	2: (* === Check loop *)
		IF NOT (MB_Lock OR MB_Start) THEN
			WHILE VarCnt<=(VARS_Max-1) AND VarSta=2 DO
				(* Check only active vars *)
				IF VARS[VarCnt].Variable<>0 THEN
					(* Check var auto-refresh on timer checks *)
					IF VARS[VarCnt].Refresh_Time>0 AND VARS[VarCnt].Refresh_Cnt=0 THEN
						VARS[VarCnt].Refresh_Cnt:=VARS[VarCnt].Refresh_Time;
						VarSta:=3;
					END_IF
					(* Check refresh for change or request *)
					CASE VARS[VarCnt].FunCode OF
						5,6,15,16: (* Write functions *)
							IF VARS[VarCnt].Variable_Size=1 THEN
								IF VARS[VarCnt].Variable^[0]<>VARS[VarCnt].Variable_Mirror THEN
									VARS[VarCnt].Variable_Mirror:=VARS[VarCnt].Variable^[0];
									VarSta:=3;
								END_IF
							ELSE
								IF VARS[VarCnt].Variable_Mirror<>0 THEN
									VARS[VarCnt].Variable_Mirror:=0;
									VarSta:=3;
								END_IF
							END_IF
						1,2,3,4: (* Write functions *)
							IF VARS[VarCnt].Variable_Mirror<>0 THEN
								VARS[VarCnt].Variable_Mirror:=0;
								VarSta:=3;
							END_IF
					END_CASE
				END_IF
				(* Process query *)
				IF VarSta=3 THEN
					MB_Lock:=TRUE;
					MB_MASTER.bUNIT_ID:=VARS[VarCnt].SlaveAddress;
					MB_MASTER.bFUNCTION_CODE:=VARS[VarCnt].FunCode;
					CASE VARS[VarCnt].FunCode OF
						16#5,16#6,16#F,16#10:
							MB_MASTER.wREAD_ADDRESS:=0;
							MB_MASTER.wREAD_QUANTITY:=0;
							MB_MASTER.wWRITE_ADDRESS:=VARS[VarCnt].FunAddress;
							MB_MASTER.wWRITE_QUANTITY:=VARS[VarCnt].Variable_Size;
							IF VARS[VarCnt].Variable_Size=200 THEN
								COPY_32SWAP16(VARS[VarCnt].Variable, ADR(MB_WRITEBUF));
							ELSIF VARS[VarCnt].Variable_Size>1 THEN
								MEMCPY(VARS[VarCnt].Variable, ADR(MB_WRITEBUF), 2*VARS[VarCnt].Variable_Size);
							ELSE
								MB_WRITEBUF[0]:=VARS[VarCnt].Variable^[0];
							END_IF
						16#1,16#2,16#3,16#4:
							MB_MASTER.wREAD_ADDRESS:=VARS[VarCnt].FunAddress;
							IF VARS[VarCnt].Variable_Size=200 THEN MB_MASTER.wREAD_QUANTITY:=2; ELSE
							  MB_MASTER.wREAD_QUANTITY:=VARS[VarCnt].Variable_Size;
							END_IF
							MB_MASTER.wWRITE_ADDRESS:=0;
							MB_MASTER.wWRITE_QUANTITY:=0;
					END_CASE
					VarRetry:=0;
					MB_Start:=TRUE;
				ELSE
					VarCnt:=VarCnt+1;
				END_IF
			END_WHILE
			(* Check loop completed -> no actions *)
			IF VarSta=2 THEN VarSta:=1; END_IF
		END_IF

	3: (* === Wait & process MB response *)
		IF NOT MB_Start THEN
			IF MB_MASTER.wERROR=0 THEN
				CASE VARS[VarCnt].FunCode OF
					1,2,3,4:
						IF VARS[VarCnt].Variable_Size=200 THEN
							COPY_32SWAP16(ADR(MB_READBUF), VARS[VarCnt].Variable);
						ELSIF VARS[VarCnt].Variable_Size>1 THEN
							MEMCPY(ADR(MB_READBUF), VARS[VarCnt].Variable, 2*VARS[VarCnt].Variable_Size);
						ELSE
							VARS[VarCnt].Variable^[0]:=MB_READBUF[0];
						END_IF
				END_CASE
				MB_Lock:=FALSE;
				(* Signal error recovery *)
				IF VARS_Alarm=TRUE AND VarCnt=VarAlarm THEN
					//LogEv(EL_Wrn,EO_MODBUS_TCP,ID,5,'');
					VARS_Alarm:=FALSE;
				END_IF
				(* Next var *)
				VarCnt:=VarCnt+1;
				VarSta:=2;
			ELSE
				IF VarRetry<2 THEN
					VarRetry:=VarRetry+1;
					MB_Start:=TRUE;
				ELSE
					MB_Lock:=FALSE;
					(* Signal error *)
					IF VARS_Alarm=FALSE THEN
						//LogEv(EL_Wrn,EO_MODBUS_TCP,ID,3,WORD_TO_STRING(MB_MASTER.wERROR));
						VARS_Alarm:=TRUE;
						VarAlarm:=VarCnt-1;
					END_IF
					(* Next var *)
					VarCnt:=VarCnt+1;
					VarSta:=2;
				END_IF
			END_IF
		END_IF

ELSE
	VarSta:=0;
END_CASE
END_ACTION

ACTION VAR_Search:
(* Search VAR with specific pointer if not found return first free VAR
	[Last VAR is not active... used as safe area...] 
*)
j:=VARS_Max;
FOR i := 0 TO VARS_Max-1 DO
	IF VARS[i].Variable=0 AND j>i THEN j:=i; END_IF
	IF VARS[i].Variable=VAR_Pointer THEN
		VAR_Cfg:=ADR(VARS[i]);
		RETURN;
	END_IF
END_FOR
VAR_Cfg:=ADR(VARS[j]);
END_ACTION

END_FUNCTION_BLOCK

// POUs/WagoLibModbus_IP_01/ETHERNET_MODBUSMASTER_TCP
FUNCTION_BLOCK ETHERNET_MODBUSMASTER_TCP
(************************************************************************************************************)
(* 750-870				                                                     		     												*)
(* Version: 0.4                                    			          														*)
(* Date: 25.03.2009                                   					          											*)
(************************************************************************************************************)
(* WAGO Kontakttechnik GmbH Hansastr. 27 32423 Minden(Westf.)									*)
(* Tel. +0049 571/887-0 Fax. +0049 571/887-0															*)
(* Author: VB																								*)
(************************************************************************************************************)
(*Description:	A  modbus master using ethernet TCP/IP protocol										*)
(*Historie: V0.4 additional errorcode wError =16#95 													*)
(*Historie: V0.3 Bugfix output wError  28.03.2008														*)
(*Historie: V0.2 release  24.02.2005																	 	*)

(*Supported modbus codes:
									0x1:	Read Coil Status 
									0x2:	Read Input Status	
									0x3:	Read Holding Registers
									0x4:	Read Multiple Register	
									0x5:	Force Single Coil
									0x6:	Write Single Register	
									0x7:	Read Exception Status				
									0x0F:	Write Multiple Coils	
									0x10:	Write Multiple Register					
									0x16:	Write Mask Register					
									0x17:	read and write multiple register								 
Error codes:
									0x01: 	Function code not supported
									0x79:	No socket available
									0x80:	Can not send modbus request
									0x81:	No response received
									0x96:	Server not available
									0x95:    Socket was "gracefully closed" by the server
									0x97:	Parameter wWRITE_QUANTITY illegal for choosen function code
									0x98: 	Response does not match to the request (overrun)
																											*)
(************************************************************************************************************)
VAR CONSTANT
	STATE_OPEN     					 :BYTE:= 0;
	STATE_TX       						 :BYTE:= 1;
	STATE_RX       					 :BYTE:= 2;
	STATE_CLOSE    					 :BYTE:= 3;
END_VAR
VAR_INPUT
	xCONNECT						:BOOL;
	strIP_ADDRESS					:STRING;
	wPORT							:WORD := 502;	 (* Port-Nr.	*)
	bUNIT_ID							:BYTE := 16#00;
	bFUNCTION_CODE				:BYTE;
	wREAD_ADDRESS				:WORD;
	wREAD_QUANTITY				:WORD;
	ptREAD_DATA					:POINTER TO WORD;
	wWRITE_ADDRESS				:WORD;
	wWRITE_QUANTITY				:WORD;
	ptSEND_DATA					:POINTER TO WORD;
	tTIME_OUT					:TIME:=t#40ms;
	tCON_WATCHDOG				:TIME:=t#1s;
END_VAR
VAR_IN_OUT
	xSEND								:BOOL;
END_VAR
VAR_OUTPUT
	xIS_CONNECTED				:BOOL;
	wERROR							:WORD;
	bRESPONSE_UNIT_ID			:BYTE := 16#00;
END_VAR

VAR
	m_State							:BYTE := 0;
	i									:INT;
	txBuffer							:ARRAY[0..1500] OF BYTE;
	rxBuffer							:ARRAY[0..1500] OF BYTE;
	txLen								:DINT;
	connected							:BOOL;
	Response							:WORD;
	ConnectionTimer					:TON;
	Socket								:DINT;
	Response_ID						:BYTE;
	Transaction_ID					:WORD;
	aux									:DINT;
	Client_OpenClose1				:Client_OpenClose;
	m_diReturn						:DINT;
	m_count							:DINT;
	m_BytesReceived					:DINT;
	ptaux								:POINTER TO ARRAY[0..1500] OF BYTE;
	pointBreak						: bool;
END_VAR

IF xConnect THEN
	(* State maschine *)
	CASE  m_State OF
	(* -------------------------------------------------------------------------*)
	STATE_OPEN:(*open connection with modbus server*)
		Client_OpenClose1(
			xOpenConnection:=xConnect ,
			xTCP:=TRUE,
			sIPaddress:=strIP_ADDRESS ,
			wPort:=wPORT ,
			diSocket:=socket ,
			xConnected=>xIS_CONNECTED );
		IF xIS_CONNECTED THEN
			m_state:=STATE_TX;
			wError:=0;
			ConnectionTimer(IN:=FALSE);
		ELSE
			ConnectionTimer(IN:=TRUE , PT:=tCON_WATCHDOG);
			IF ConnectionTimer.Q THEN(*watchdog time expired*)
				wError:=16#96;(*server not available*)
				ConnectionTimer(IN:=FALSE);
				m_state:=state_close;
			END_IF
		END_IF
	(* -------------------------------------------------------------------------*)
	STATE_TX:(*process modbus request*)
		if bUNIT_ID = 9 then
			pointBreak := TRUE;
		end_if
		if wWRITE_ADDRESS = 319 then
			pointBreak := TRUE;
		end_if
		IF xSend THEN
			aux:=ModbusRequest(
				bUNIT_ID:=bUNIT_ID,
				bFUNCTION_CODE:=bFUNCTION_CODE,
				wREAD_ADDRESS:=wREAD_ADDRESS,
				wREAD_QUANTITY:=wREAD_QUANTITY,
				ptREAD_DATA:=ptREAD_DATA,
				wWRITE_ADDRESS:=wWRITE_ADDRESS,
				wWRITE_QUANTITY:=wWRITE_QUANTITY,
				ptSEND_DATA:=ptSEND_DATA,
				TRANSACTION_ID:=Transaction_ID,
				RESPONSE:=Response,
				TelegrammData:=txBuffer);

			IF aux>0 THEN (*modbus request data valid*)
				m_diReturn := SysSockSend(diSocket := Socket, pbyBuffer := ADR(txBuffer[0]), diBufferSize := aux,diFlags := 0);
				CASE m_diReturn OF
				-1:	(* ERROR *)
					ConnectionTimer(IN:=TRUE , PT:=tTIME_OUT);
					IF ConnectionTimer.Q THEN(*watchdog time expired*)
						wError:=16#80;(*could not send modbus request*)
						m_state:=STATE_CLOSE;
						ConnectionTimer(IN:=FALSE , PT:=tTIME_OUT);
					END_IF
				0: (* socket was "gracefully closed" *)
					m_State := STATE_CLOSE;
				ELSE (* succesful *)
					m_count:=m_count+m_diReturn;
					IF m_count>=aux THEN
						ConnectionTimer(IN:=FALSE);
						m_State := STATE_RX;
						m_count:=0;
					END_IF
				END_CASE
			ELSE(*modbus request data faulty*)
					xSend:=FALSE;
					m_State:=STATE_TX;
					wError:=DINT_TO_WORD(-1*aux) ;
			END_IF
		END_IF
	(* -------------------------------------------------------------------------*)
	STATE_RX: (* process modbus response *)
			m_BytesReceived := SysSockRecv(diSocket := Socket,
												pbyBuffer 	:= ADR(rxBuffer),		(* Address of receive buffer *)
												diBufferSize:= SIZEOF(rxBuffer),
												diFlags		:= 0);

			CASE m_BytesReceived OF
			-1:	(* No data available or error occured *)
				ConnectionTimer(IN:=TRUE , PT:=tTIME_OUT);
				IF ConnectionTimer.Q THEN(*watchdog time expired*)
					wError:=16#81;(*no response received*)
					xSend:=FALSE;(*V0.4 added*)
					m_State:=STATE_CLOSE;
					ConnectionTimer(IN:=FALSE , PT:=tTIME_OUT);
				END_IF;
			0: (* socket was "gracefully closed"  *)
				m_State:=STATE_CLOSE;
				wError:=16#95;(*V0.4 added*)
				xSend:=FALSE;(*V0.4 added*)
			ELSE (* succesful *)
				IF m_BytesReceived = Response THEN (* Answer is complete *)
					bRESPONSE_UNIT_ID := rxBuffer[6];
					IF (m_BytesReceived = 9) AND (rxBuffer[7] AND 16#80) <> 16#00 THEN  (* Error Message *)
						wError := rxBuffer[8];
					ELSE
						CASE BYTE_TO_INT(bFUNCTION_CODE) OF

							READ_COILS, READ_INPUT_DISCRETES :
									ptaux:=ptRead_Data;
									FOR i := 9 TO DINT_TO_INT(m_BytesReceived)-1 DO
										ptaux^[i-9] := rxBuffer[i];
									END_FOR

							READ_MULTIPLE_REGISTERS, READ_INPUT_REGISTERS, READ_WRITE_REGISTERS :
									ptaux:=ptRead_Data;
									FOR i := 9 TO DINT_TO_INT( m_BytesReceived)-1 BY 2 DO
										ptaux^[i-9] := rxBuffer[i];
										ptaux^[i-8] := rxBuffer[i+1];
									END_FOR
						END_CASE
						IF rxBuffer[7] = READ_EXCEPTION_STATUS THEN
							ptaux:=ptRead_Data;
							ptaux^[0] := rxBuffer[i-1];
						END_IF
						wError := 16#00;
					END_IF
				ELSIF m_BytesReceived >= 9 THEN  (* Is Error-Message ? *)
					IF (rxBuffer[7] AND 16#80) <> 16#00 THEN  (* Error Message *)
						bRESPONSE_UNIT_ID := rxBuffer[6];
						wError := rxBuffer[8];
					ELSE   (* OVERRUN *)
						wError := 16#98; (* OVERRUN *)
					END_IF
				END_IF
				ConnectionTimer(IN:=FALSE);
				m_State:=STATE_TX;
				xSend:=FALSE;
			END_CASE
	(* -------------------------------------------------------------------------*)
	STATE_CLOSE:
		Client_OpenClose1(
					xOpenConnection:=FALSE,
					xTCP:=TRUE,
					sIPaddress:=strIP_ADDRESS ,
					wPort:=wPORT ,
					xConnected=>xIS_CONNECTED ,
					diSocket:=Socket );
			IF Client_OpenClose1.xConnected=FALSE THEN
				m_State:=STATE_OPEN;
			END_IF

	END_CASE
(**************************************************************************************)

ELSE(*close connection*)
	xSend:=FALSE;
	Client_OpenClose1(
		xOpenConnection:=FALSE,
		xTCP:=TRUE,
		sIPaddress:=strIP_ADDRESS ,
		wPort:=wPORT ,
		xConnected=>xIS_CONNECTED ,
		diSocket:=Socket );
	m_State:=STATE_OPEN;
	ConnectionTimer(IN:=FALSE);
	wError:=0;	(*V0.3*)
END_IF

END_FUNCTION_BLOCK

// POUs/WagoLibModbus_IP_01/ModbusRequest
FUNCTION ModbusRequest : DINT
(************************************************************************************************************)
(* Version: 0.3                                    			          														*)
(* Date: 02.04.2013                                   					          											*)
(************************************************************************************************************)
(* WAGO Kontakttechnik GmbH Hansastr. 27 32423 Minden(Westf.)									*)
(* Tel. +0049 571/887-0 Fax. +0049 571/887-0															*)
(* Author: VB																								*)
(*Historie:																									*)
(*Version 0.3: FC22 implemented (UU)																	*)
(*Version 0.2: Cast operator DINT_TO_BYTE replaced by WORD_TO_BYTE due to compiler 2.3.7.1	*)
(*Version 0.1: Release																					*)
(************************************************************************************************************)
(*Description:	Building a modbus request for the following function codes:
									0x1:	Read Coil Status 
									0x2:	Read Input Status	
									0x3:	Read Holding Registers
									0x4:	Read Multiple Register	
									0x5:	Force Single Coil
									0x6:	Write Single Register	
									0x7:	Read Exception Status				
									0x0F:	Write Multiple Coils	
									0x10:	Write Multiple Register					
									0x16:   Write Mask Register
									0x17:	read and write multiple register								 *)
VAR_INPUT
	bUNIT_ID						:	BYTE := 16#00;
	bFUNCTION_CODE			:	BYTE;
	wREAD_ADDRESS			:	WORD;
	wREAD_QUANTITY			:	WORD;
	ptREAD_DATA				:	POINTER TO ARRAY[0..1500] OF BYTE;
	wWRITE_ADDRESS			:	WORD;
	wWRITE_QUANTITY			:	WORD;
	ptSEND_DATA				:	POINTER TO ARRAY[0..1500] OF BYTE;
END_VAR
VAR_IN_OUT
	TRANSACTION_ID			:	WORD;
	RESPONSE					:	WORD;
	TelegrammData				:	ARRAY[0..1500] OF BYTE;
END_VAR
VAR
	i								: 	INT;
END_VAR


				Transaction_ID := Transaction_ID + 1;
				(* ---- H E A D E R ------------------------------------------------------------------- *)
				TelegrammData[0] := WORD_TO_BYTE(SHR(Transaction_ID,8)); 	(* TRANSACTION-ID HI-Byte 	*)
				TelegrammData[1] := WORD_TO_BYTE(Transaction_ID);			(* TRANSACTION-ID LO-Byte	*)
				TelegrammData[2] := 16#00;									(* PROTOKOLL-ID HI-Byte 	*)
				TelegrammData[3] := 16#00;									(* PROTOKOLL-ID LO-Byte 	*)

				TelegrammData[4] := 16#00;
				TelegrammData[5] := 16#00;									(* Laenge 					*)

				TelegrammData[6] := bUNIT_ID;								(* UNIT						*)
				TelegrammData[7] := bFUNCTION_CODE;							(* FUNCTION-CODE			*)
				(*----- END OF HEADER ------------------------------------------------------------------*)

				(* --------------------------------------------------- *)
				CASE BYTE_TO_INT(bFUNCTION_CODE) OF
					READ_COILS, READ_INPUT_DISCRETES :
						(**** 01 Read Coil Status /  02 Read Input Status **********************)
						TelegrammData[8] := WORD_TO_BYTE(SHR(wREAD_ADDRESS,8));
						TelegrammData[9] := WORD_TO_BYTE(wREAD_ADDRESS);
						TelegrammData[10] := WORD_TO_BYTE(SHR(wREAD_QUANTITY,8));
						TelegrammData[11] := WORD_TO_BYTE(wREAD_QUANTITY);
						TelegrammData[5] := 16#06;						(* Laenge 						*)
						IF (wREAD_QUANTITY >= 0) THEN
							Response :=	SHR(wREAD_QUANTITY + 7,3)  + 9; (* # *)
						END_IF
						ModbusRequest:=12;(*Länge des Telegramms*)
					3,4:(*READ_MULTIPLE_REGISTERS, READ_INPUT_REGISTERS :*)
						(**** 03 Read Holding Registers / 04 Read Input Registers ***********)
						TelegrammData[8] := WORD_TO_BYTE(SHR(wREAD_ADDRESS,8));
						TelegrammData[9] := WORD_TO_BYTE(wREAD_ADDRESS);
						TelegrammData[10] := WORD_TO_BYTE(SHR(wREAD_QUANTITY,8));
						TelegrammData[11] := WORD_TO_BYTE(wREAD_QUANTITY);
						TelegrammData[5] := 16#06;						(* Laenge 						*)
						Response :=wREAD_QUANTITY * 2 + 9; (* # *)
						ModbusRequest:=12;(*Länge des Telegramms*)
					WRITE_COIL :
						(**** 05 Force Single Coil *******************************************)
						TelegrammData[8] := WORD_TO_BYTE(SHR(wWRITE_ADDRESS,8));
						TelegrammData[9] := WORD_TO_BYTE(wWRITE_ADDRESS);
						IF (ptSEND_DATA^[0] AND 16#01) = 16#01 THEN
							TelegrammData[10] := 16#FF;	(* Einschalten *)
						ELSE
							TelegrammData[10] := 16#00;	(* Ausschalten *)
						END_IF
						TelegrammData[11] := 16#00;
						TelegrammData[5] := 16#06;						(* Laenge 						*)
						Response :=	12; (* # *)
						ModbusRequest:=12;(*Länge des Telegramms*)
					WRITE_SINGLE_REGISTER :
						(**** 06 Preset Single Register *************************************)
						TelegrammData[8] := WORD_TO_BYTE(SHR(wWRITE_ADDRESS,8));
						TelegrammData[9] := WORD_TO_BYTE(wWRITE_ADDRESS);
						TelegrammData[10] := ptSEND_DATA^[0];
						TelegrammData[11] := ptSEND_DATA^[1];
						TelegrammData[5] := 16#06;						(* Laenge 						*)
						Response :=	12; (* # *)
						ModbusRequest:=12;(*Länge des Telegramms*)
					READ_EXCEPTION_STATUS :
						(**** 07 Read Exception Status ****************************)
						TelegrammData[5] := 16#02;						(* Laenge 						*)
						Response :=	9; (* # *)
						ModbusRequest:=8;(*Länge des Telegramms*)
					FORCE_MULTIPLE_COILS :
						(**** 0F Force Multiple Coils 		*)
						TelegrammData[8] := WORD_TO_BYTE(SHR(wWRITE_ADDRESS,8));
						TelegrammData[9] := WORD_TO_BYTE(wWRITE_ADDRESS);
						IF (wWRITE_QUANTITY <= 2040) AND (wWRITE_QUANTITY >= 0) THEN
							TelegrammData[10] := WORD_TO_BYTE(SHR(wWRITE_QUANTITY,8));  	(*Quantity of coils high *)
							TelegrammData[11] := WORD_TO_BYTE(wWRITE_QUANTITY);			(*Quantity of coils low   *)
							(*** Byte Counter calculate ***)
							TelegrammData[12] := WORD_TO_BYTE((wWRITE_QUANTITY + 7) / 8);

							(**************************************************************************************************)
							FOR i := 0 TO TelegrammData[12]  DO
								TelegrammData[i + 13] := ptSend_DATA^[i];
							END_FOR
							TelegrammData[5] := 7+TelegrammData[12];						(* Laenge 						*)
							Response :=	12; (* # *)
							ModbusRequest:=TelegrammData[12]+13;(*Länge des Telegramms*)
						ELSE
							ModbusRequest:=-97;(* ILLEGAL NUMBER OF POINTS *)
							(*wError := 16#97;	*)(* ILLEGAL NUMBER OF POINTS *)
						END_IF

				WRITE_MULTIPLE_REGISTERS :
						(**** 10 Preset Multiple Registers 	*)
						TelegrammData[8] := WORD_TO_BYTE(SHR(wWRITE_ADDRESS,8));
						TelegrammData[9] := WORD_TO_BYTE(wWRITE_ADDRESS);
						IF (wWRITE_QUANTITY <= 127) AND (wWRITE_QUANTITY >= 0) THEN
							TelegrammData[10] := WORD_TO_BYTE(SHR(wWRITE_QUANTITY,8));  	(*Number of register high *)
							TelegrammData[11] := WORD_TO_BYTE(wWRITE_QUANTITY);			(*Number of register low *)
							(*** Byte Counter calculate ***)
							TelegrammData[12] := WORD_TO_BYTE(wWRITE_QUANTITY * 16#0002);
							(**************************************************************************************************)
							FOR i:= 0 TO (wWRITE_QUANTITY-1) DO
								TelegrammData[14+2*i]:= ptSEND_DATA^[2*i+1];
								TelegrammData[13+2*i]:= ptSEND_DATA^[2*i];
							END_FOR
							TelegrammData[5] := TelegrammData[12]+7;						(* Laenge 						*)
							Response :=	12;
							ModbusRequest := TelegrammData[12]+13;
						ELSE
							ModbusRequest:=-97;
							(*wError := 16#97;	*)(* ILLEGAL NUMBER OF POINTS *)
						END_IF

				READ_WRITE_REGISTERS :
						(**** 17 Read/Write Multiple Registers 	*)
						(*** READ ****)
						TelegrammData[8] := WORD_TO_BYTE(SHR(wREAD_ADDRESS,8));
						TelegrammData[9] := WORD_TO_BYTE(wREAD_ADDRESS);
						TelegrammData[10] := WORD_TO_BYTE(SHR(wREAD_QUANTITY,8));
						TelegrammData[11] := WORD_TO_BYTE(wREAD_QUANTITY);
						(*** WRITE ****)
						TelegrammData[12] := WORD_TO_BYTE(SHR(wWRITE_ADDRESS,8));
						TelegrammData[13] := WORD_TO_BYTE(wWRITE_ADDRESS);
						TelegrammData[14] := WORD_TO_BYTE(SHR(wWRITE_QUANTITY,8));  	(*Number of register high *)
						TelegrammData[15] := WORD_TO_BYTE(wWRITE_QUANTITY);				(*Number of register low *)
						(*** Byte Counter calculate ***)
						TelegrammData[16] := WORD_TO_BYTE(wWRITE_QUANTITY * 16#0002);
						(***********************************************************************)

						FOR i:= 0 TO (wWRITE_QUANTITY-1) DO
							TelegrammData[18+2*i]:= ptSEND_DATA^[2*i];
							TelegrammData[17+2*i]:= ptSEND_DATA^[2*i+1];
						END_FOR
						TelegrammData[5] := TelegrammData[16]+11;						(* Laenge 						*)
						Response :=wREAD_QUANTITY * 2 + 9;
						ModbusRequest := TelegrammData[16]+17;

				(*=== INSERT NEW FC22 -> 02.04.2013 UU =====================================*)
				WRITE_MASK_REGISTER : (* new function code FC22 -> 02.04.2013 UU *)
						(**** 10 Preset Multiple Registers 	*)
						TelegrammData[8] := WORD_TO_BYTE(SHR(wWRITE_ADDRESS,8));
						TelegrammData[9] := WORD_TO_BYTE(wWRITE_ADDRESS);
						IF (wWRITE_QUANTITY = 2)  THEN

							TelegrammData[10] := ptSEND_DATA^[0];  	(* AND-Mask H-Byte *)
							TelegrammData[11] := ptSEND_DATA^[1];  	(* AND-Mask L-Byte *)

							TelegrammData[12] := ptSEND_DATA^[2];  	(* OR-Mask H-Byte *)
							TelegrammData[13] := ptSEND_DATA^[3];  	(* OR-Mask L-Byte *)

							TelegrammData[5]  := 8;					(* Laenge 			*)
							Response 		  := 14;	(* expected response length *)
							ModbusRequest 	  := 14;	(* Frame length *)

						ELSE
							ModbusRequest:=-97;
							(*wError := 16#97;	*)(* ILLEGAL NUMBER OF POINTS *)
						END_IF
				(*==========================================================================*)

		(**************************************************************************************************)
				ELSE
						ModbusRequest:=-1;
						(*wError := 16#01;	*)(* ILLEGAL FUNCTION *)
				END_CASE;

END_FUNCTION

// POUs/WagoLibModbus_IP_01/Client_OpenClose
FUNCTION_BLOCK Client_OpenClose
(************************************************************************************************************)
(* 750-870				                                                     		     												*)
(* Version: 0.6                                    			          														*)
(* Date: 16.01.13                                   					          												*)
(************************************************************************************************************)
(* WAGO Kontakttechnik GmbH Hansastr. 27 32423 Minden(Westf.)									*)
(* Tel. +0049 571/887-0 Fax. +0049 571/887-0															*)
(* Author: VB																								*)
(************************************************************************************************************)
(*Description:	A  client open block																      		*)
(*Historie: V0.6 Bugfix close in case timeout 	16.01.13												*)
(*Historie: V0.5 Improvement FW13	26.05.08															*)
(*Historie: V0.4 Push bit added	17.12.07																*)
(*Historie: V0.3 Changes socket handle zero													 	      	*)
(*Historie: V0.2 Release		21.01.05															 	       *)
(************************************************************************************************************)
VAR CONSTANT
	STATE_CREATE     				: BYTE:= 0;
	STATE_CONNECT     				: BYTE:= 10;
	STATE_IDLE      					: BYTE:= 20;
	STATE_CLOSE    					: BYTE:= 40;
	CONNECT_WATCHDOG_TIME	: TIME:=t#10s;
END_VAR

VAR_INPUT
	xOpenConnection					: BOOL;
	xTCP								: BOOL;(*True open a TCP socket; False:open a UDP socket*)
	sIPaddress						: STRING(80); //GIURE modifica per evitare warning (valeva 16 IP:= xxx.yyy.zzz.ttt)
	wPort								: WORD;
END_VAR
VAR_IN_OUT
	diSocket							: DINT;
END_VAR
VAR_OUTPUT
	xConnected						: BOOL;
END_VAR
(* ErrorCodes -----------------------------------------
	-1 => No socket descriptor available 
	-4 => socket supports only blocking mode 
	-6 => connection could not be established 
	16#8005 => SysSockClose() returns FALSE 
    	16#8006 => SysSockConnect() fails
------------------------------------------------------------*)

VAR
	m_State								: BYTE := 0;
	m_Socket								: DINT;
	m_AddressInfo						: SOCKADDRESS;
	m_BytesReceived						: DINT;
	m_diReturn							: DINT;
	m_xReturn							: BOOL;
	m_IoCtlParameter  					: DINT:= 1; (* IOCTL-Parameter for non-blocking mode of sockets *)
	i										: INT;
	T_Connect							: TON;
	m_count								:DINT;
	diOption							:DINT:=1;
END_VAR

IF xOpenConnection THEN
	(* State maschine *)
	CASE  m_State OF

	(* -------------------------------------------------------------------------*)
	STATE_CREATE:
			(* create socket descriptor*)
		IF xTCP THEN
			m_Socket := SysSockCreate(diAddressFamily	:= SOCKET_AF_INET,
													 diType		:= SOCKET_STREAM,
													 diProtocol := SOCKET_IPPROTO_TCP);
			IF m_Socket >= 0 THEN(*create was successful*)

(*V0.4*)		(* change  socket mode  to set push bit with each telegramm *)
				SysSockSetOption(
					diSocket:=m_Socket,
					diLevel:=6,
					diOption:=SOCKET_TCP_NODELAY,
					pOptionValue:=ADR(diOption),
					diOptionLength:=SIZEOF(diOption));


(***********)
				(* change  socket mode  to none blocking *)
				m_diReturn := SysSockIoctl( m_Socket, SOCKET_FIONBIO, ADR(m_IoCtlParameter));
				//IF m_diReturn <> 0 THEN
					m_AddressInfo.sin_family := SOCKET_AF_INET;
					m_AddressInfo.sin_port := SysSockNtohs(wPort);
					m_AddressInfo.sin_addr :=  SysSockInetAddr(sIPaddress) ;
					m_State := STATE_CONNECT;
				//ELSE
					//	diSocket := -4;  (* socket supports only blocking mode*)
					//	m_State := STATE_IDLE;
				//END_IF

			ELSE(*create failed*)
					diSocket := -1;  (* no socket descriptor available *)
					m_State := STATE_IDLE;
			END_IF
		ELSE(*UDP*)
			m_Socket := SysSockCreate(diAddressFamily	 := SOCKET_AF_INET,
											 		diType		:= SOCKET_DGRAM,
													 diProtocol := SOCKET_IPPROTO_UDP);
			IF m_Socket >= 0 THEN(*create was succeful*)
				(* change  socket mode  to none blocking *)
				m_diReturn := SysSockIoctl( m_Socket, SOCKET_FIONBIO, ADR(m_IoCtlParameter));
				m_State := STATE_IDLE;
				diSocket:=m_socket;
				xConnected:=TRUE;
			ELSE
				diSocket := -1;  (* no socket descriptor available *)
				m_State := STATE_IDLE;
			END_IF

		END_IF
	(* -------------------------------------------------------------------------*)
	STATE_CONNECT: (* try to connect with server *)
		T_Connect(IN:=TRUE , PT:=CONNECT_WATCHDOG_TIME);(*activate watchdog for establishing connection to a server*)
		m_xReturn := SysSockConnect ( m_Socket, ADR(m_AddressInfo),  SIZEOF(m_AddressInfo));
		IF m_xReturn THEN (* succesful *)
			diSocket:=m_socket;
			m_State := STATE_IDLE;
			xConnected:=TRUE;
			T_Connect(IN:=FALSE);
			(*V0.4*)	(* change  socket mode  to set push bit with each telegramm *)
			SysSockSetOption(
				diSocket:=m_Socket,
				diLevel:=6,
				diOption:=SOCKET_TCP_NODELAY,
				pOptionValue:=ADR(diOption),
				diOptionLength:=SIZEOF(diOption));
		ELSE
			IF T_Connect.Q THEN
				diSocket := -6;  (* connect fails *)
				xConnected:=FALSE;
				T_Connect(IN:=FALSE);
				m_State := STATE_IDLE;
				IF m_Socket >=0 THEN
					SysSockClose( m_Socket);
					m_Socket := -1;		(*V0.6*)
				END_IF
			ELSE
				m_State := STATE_CONNECT;(*client still  tries to set up connection*)
			END_IF
		END_IF

	(* -------------------------------------------------------------------------*)
	STATE_IDLE: (* error handling *)
	;

	END_CASE

ELSE(*close connection*)
	IF m_Socket >= 0 THEN
		SysSockClose( m_Socket);
		m_Socket := -1;		(*V0.5*)
		diSocket := -1;
	END_IF

	m_State := STATE_CREATE;
	xConnected:=FALSE;
END_IF

END_FUNCTION_BLOCK

// POUs/Plant_Objects/obj_CRON
FUNCTION_BLOCK obj_CRON
(* === CRONOGRAFO STANDARD ===
   v1.0[16/04/05] - Versioning
*)
VAR_INPUT
	(* Settings *)
	ID			: BYTE;		(* Index of instanced object *)

	InitOK		: BOOL;
	Alarm		: BOOL;
	Warning		: BOOL;

	Profile		: typ_Cron_Profile; 				(* Profilo attivo *)
	ProfileNr	: BYTE;								(* Indice profilo attivo *)
	CalendarIdx : WORD;								(* Indice calendario attivo *)
	Jolly		: ARRAY[0..9] OF typ_Cron_Jolly;	(* Jolly attivi *)

	SET_POINT		: INT;	//GIURE ver 21
	(* Status *)
	STAT_LOG		: BYTE; //GIURE ver 21

END_VAR
VAR_IN_OUT
END_VAR
VAR_OUTPUT
	SetPoint		: INT;
	(* Status *)
	Status_Log		: BYTE;
	Status_Vis 		: DWORD;
END_VAR
VAR
	Buf: 	ARRAY[0..512] OF BYTE;
	hFile		: RTS_IEC_HANDLE;
	hRes		: RTS_IEC_RESULT;
	sFile: 	STRING;
	sFile2: STRING;

	i:		WORD;
	t1:		DWORD;
	t2:		BOOL;

END_VAR

(* Check initialization *)
IF NOT 
	InitOK 
THEN 
	Init(); 
END_IF

(* Chrono *)
IF CalendarIdx<>Sys.Time_CT_Day THEN DB_Load(); END_IF
SetPoint:=Profile.Setpoint[Sys.Time_CT_Quarter];

(* Check jolly *)
FOR i := 0 TO 9 DO
	IF ( DT_TO_DWORD(Jolly[i].Start)>0  AND Jolly[i].End>Jolly[i].Start AND
	     Jolly[i].Start<=Sys.Time_CT_DT AND Jolly[i].End>Sys.Time_CT_DT ) THEN
			SetPoint:=Jolly[i].Temp;
	END_IF
END_FOR


(* Status color *)
   IF Alarm   THEN Status_Log:=2; Status_Vis:=16#2020F0;
ELSIF Warning THEN Status_Log:=1; Status_Vis:=16#20F0F0;
              ELSE Status_Log:=0; Status_Vis:=16#20F020;
			  END_IF

ACTION DB_Create:
(*(* Check presence of previous year *)
sFile2:=REPLACE(STR1:=sFile, STR2:=WORD_TO_STRING(Sys.Time_Year-1), L:=4, P:=LEN(FilesPath)+1);
hFile:=SysFileOpen(sFile2, AM_READ, ADR(hRes));
IF hFile<>RTS_INVALID_HANDLE THEN
	(* Check file version and close *)
	SysFileRead(hFile, ADR(Buf), 1, ADR(hRes));
	SysFileClose(hFile);
END_IF
IF hFile<>RTS_INVALID_HANDLE AND Buf[0]=1 THEN
	(* Copy file *)
	SysFileCopy(sFile, sFile2);
ELSE*)
	(* Create empty file *)
	hFile:=SysFileOpen(sFile, AM_WRITE, ADR(hRes));
	MEMCLR(pDestinationAddress:=ADR(Buf), BytesToClear:=SIZEOF(Buf));
	FOR i := 0 TO 10239 BY 512 DO
		SysFileWrite(hFile, ADR(Buf), 512, ADR(hRes));
	END_FOR
	Buf[0]:=1;
	SysFileSetPos(hFile, 0);
	SysFileWrite(hFile, ADR(Buf), 1, ADR(hRes));
	SysFileClose(hFile);
//END_IF
END_ACTION

ACTION DB_Load:
DB_SetName();

(* Open data file *)
hFile:=SysFileOpen(sFile, AM_READ, ADR(hRes));

(* File not found *)
IF hFile=RTS_INVALID_HANDLE THEN
	Warning:=TRUE;
	LogEv(EL_Wrn,EO_CRON,ID,1,'No_data_file');
	DB_Create();
	(* Reopen file *)
	hFile:=SysFileOpen(sFile, AM_READ, ADR(hRes));
	IF hFile=RTS_INVALID_HANDLE THEN
		Alarm:=TRUE;
		LogEv(EL_Alarm,EO_CRON,ID,3,'Filesystem_error');
		RETURN;
	END_IF
END_IF

(* Check version *)
SysFileRead(hFile, ADR(Buf), 1, ADR(hRes));
IF Buf[0]<>1 THEN
	IF NOT Alarm THEN
		Alarm:=TRUE;
		LogEv(EL_Alarm,EO_CRON,ID,2,'Bad_data_version');
	END_IF
	SysFileClose(hFile);
	RETURN;
END_IF

(* Read Jolly data *)
SysFileSetPos(hFile, 512);
SysFileRead(hFile, ADR(Jolly), SIZEOF(Jolly), ADR(hRes));
(* Read active profile index *)
CalendarIdx:=Sys.Time_CT_Day;
SysFileSetPos(hFile, (1024+4*CalendarIdx));
SysFileRead(hFile, ADR(ProfileNr), SIZEOF(ProfileNr), ADR(hRes));
(* Read active profile *)
SysFileSetPos(hFile, (3072+512*ProfileNr));
SysFileRead(hFile, ADR(Profile), SIZEOF(Profile), ADR(hRes));

(* Close file and validate data *)
SysFileClose(hFile);
END_ACTION

ACTION DB_SetName:
(* Create current filename 'yyyyCRnn.DAT' *)
sFile:=CONCAT(ConfPath,WORD_TO_STRING(Sys.Time_Year));
sFile:=CONCAT(STR1:=sFile, STR2:='CR');
IF ID<10 THEN
sFile:=CONCAT(STR1:=sFile, STR2:='0');
END_IF
sFile:=CONCAT(STR1:=sFile, STR2:=BYTE_TO_STRING(ID));
sFile:=CONCAT(STR1:=sFile, STR2:='.DAT');
END_ACTION

ACTION Init:
DB_Load();
InitOK:=TRUE;
END_ACTION

ACTION AddLogData:
//Genera la stringa di log dei cronografi	//GIURE ver 21
//Logger.s1:=INSERT('&CRON=',BYTE_TO_STRING(ID),5);
Logger.s1:=INSERT('&CRON=',WORD_TO_STRING(ID),5);
IF ID<10 THEN Logger.s1:=INSERT(Logger.s1,'0',5); END_IF

Logger.s1:=CONCAT(Logger.s1,INT_TO_STRING(SET_POINT));		
Logger.s1:=CONCAT(Logger.s1,';');
Logger.s1:=CONCAT(Logger.s1,BYTE_TO_STRING(STAT_LOG));
ADDSTRING(ADR(Logger.TData), ADR(Logger.s1), Logger.TLen);
END_ACTION

END_FUNCTION_BLOCK

// POUs/Plant_Objects/obj_CRON_EDITOR
FUNCTION_BLOCK obj_CRON_EDITOR
(* === EDITOR CRONOGRAFO ===
   v1.0[16/04/05] - Versioning
*)
VAR_INPUT

	(* Common selections *)
	CN_Sel:			BYTE:=1;
	CN_Act:			BYTE;
	CN_YSel:		WORD:=2015;
	CN_YAct:		WORD;

	(* Profile editor *)
	PR_Sel: 		BYTE:=1;
	PR_Act:			BYTE;
	PR_TT:			REAL;
	PR:				typ_Cron_Profile;
	(* Profile signals *)
	PR_Load:		BOOL;
	PR_Save:		BOOL;

	(* Calendar editor *)
	CA_Sel:			BYTE:=1; (* Calendar month selected *)
	CA_Act:			BYTE;    (* Calendar month active *)
	CA_DayF:		BYTE:=0;
	CA_DayL:		BYTE:=31;
	CA_TPR:			BYTE;
	CA:				typ_Cron_Calendar; (* Only used for first 32 entries *)
	(* Calendar signals *)
	CA_Load:		BOOL;
	CA_Save:		BOOL;

	(* Jolly editor *)
	JL:				ARRAY[0..9] OF typ_Cron_Jolly;
	(* Jolly signals *)
	JL_Load:		BOOL;
	JL_Save:		BOOL;

END_VAR
VAR_OUTPUT
	Message		: STRING;
END_VAR
VAR
	sFileName	: STRING;
	hMode		: ACCESS_MODE;
	hFile		: RTS_IEC_HANDLE;
	hRes		: RTS_IEC_RESULT;

	i			: WORD;
	ver			: BYTE;
	r1			: BOOL;
	r2			: DWORD;

END_VAR

IF PR_Load 
	THEN 
		PR_Load_Exe(); 
		PR_Load:=FALSE; 
END_IF
IF PR_Save 
	THEN 
		PR_Save_Exe(); PR_Save:=FALSE; 
END_IF
IF CA_Load 
THEN 
	CA_Load_Exe(); CA_Load:=FALSE; 
END_IF
IF CA_Save 
THEN 
	CA_Save_Exe(); CA_Save:=FALSE; 
END_IF
IF JL_Load 
	THEN 
	JL_Load_Exe(); JL_Load:=FALSE; 
END_IF
IF JL_Save 
	THEN 
	JL_Save_Exe(); JL_Save:=FALSE; 
END_IF

ACTION CA_Load_Exe:
hMode:=AM_READ;
FileOpen();

IF hFile<>RTS_INVALID_HANDLE THEN

	(* Read calendar month *)
	FOR i := 0 TO 31 DO
		SysFileSetPos(hFile, (1024 + ((CA_Sel-1)*32 + i)*4) );
		SysFileRead(hFile, ADR(CA.Profile[i]), 1, ADR(hRes));
	END_FOR

	(* Close file *)
	SysFileClose(hFile);

	(* Validate data *)
	CA_Act :=CA_Sel;
	CN_Act :=CN_Sel;
	CN_YAct:=CN_YSel;

	Message:='Calendar load OK';

END_IF
END_ACTION

ACTION CA_Save_Exe:
hMode:=AM_READ_PLUS;
FileOpen();

IF hFile<>RTS_INVALID_HANDLE THEN

	(* Write calendar month *)
	FOR i := 0 TO 31 DO
		SysFileSetPos(hFile, (1024 + ((CA_Sel-1)*32 + i)*4) );
		SysFileWrite(hFile, ADR(CA.Profile[i]), 1, ADR(hRes));
	END_FOR

	(* Close file *)
	SysFileClose(hFile);

	Message:='Calendar save OK';

END_IF
END_ACTION

ACTION FileOpen:
(* Create current filename 'yyyyCRnn.DAT' *)
sFileName:=CONCAT(ConfPath,WORD_TO_STRING(CN_YSel));
sFileName:=CONCAT(STR1:=sFileName, STR2:='CR');
IF CN_Sel<10 THEN
sFileName:=CONCAT(STR1:=sFileName, STR2:='0');
END_IF
sFileName:=CONCAT(STR1:=sFileName, STR2:=BYTE_TO_STRING(CN_Sel));
sFileName:=CONCAT(STR1:=sFileName, STR2:='.DAT');

(* Check file version and size! *)
(* ... *)

(* Open data file *)
hFile:=SysFileOpen(sFileName,AM_READ,ADR(hRes));

(* File not found *)
IF hFile=RTS_INVALID_HANDLE THEN
	Message:='File not found';
	RETURN;
END_IF

(* Close file *)
SysFileClose(hFile);

(* Open data file *)
hFile:=SysFileOpen(sFileName,hMode,ADR(hRes));
END_ACTION

ACTION JL_Load_Exe:
hMode:=AM_READ;
FileOpen();

IF hFile<>RTS_INVALID_HANDLE THEN

	(* Read jolly *)
	SysFileSetPos(hFile, 512);
	SysFileRead(hFile, ADR(JL), SIZEOF(JL), ADR(hRes));

	(* Close file *)
	SysFileClose(hFile);

	(* Validate data *)
	CN_Act:=CN_Sel;
	CN_YAct:=CN_YSel;

	Message:='Jolly load OK';

END_IF
END_ACTION

ACTION JL_Save_Exe:
hMode:=AM_READ_PLUS;
FileOpen();

IF hFile<>RTS_INVALID_HANDLE THEN

	(* Write selected profile *)
	SysFileSetPos(hFile, 512);
	SysFileWrite(hFile, ADR(JL), SIZEOF(JL), ADR(hRes));

	(* Close file *)
	SysFileClose(hFile);

	Message:='Jolly save OK';

END_IF
END_ACTION

ACTION PR_Load_Exe:
hMode:=AM_READ;
FileOpen();

IF hFile<>RTS_INVALID_HANDLE THEN

	(* Read selected profile *)
	SysFileSetPos(hFile, (3072 + 512*PR_Sel));
	SysFileRead(hFile, ADR(PR), SIZEOF(PR), ADR(hRes));

	(* Close file *)
	SysFileClose(hFile);

	(* Validate data *)
	PR_Act:=PR_Sel;
	CN_Act:=CN_Sel;
	CN_YAct:=CN_YSel;

	Message:='Profile load OK';

END_IF
END_ACTION

ACTION PR_Save_Exe:
hMode:=AM_READ_PLUS;
FileOpen();

IF hFile<>RTS_INVALID_HANDLE THEN

	(* Write selected profile *)
	SysFileSetPos(hFile, (3072 + 512*PR_Sel));
	SysFileWrite(hFile, ADR(PR), SIZEOF(PR), ADR(hRes));

	(* Close file *)
	SysFileClose(hFile);

	Message:='Profile save OK';

END_IF
END_ACTION

END_FUNCTION_BLOCK

// POUs/Plant_Objects/obj_ASI
FUNCTION_BLOCK obj_ASI
(* === ASi INTERFACE ===
   v0.0[21/05/15] - Creation
*)
VAR_INPUT
	(* Settings *)
	ID				: BYTE;
	Refresh_Period	: TIME:=T#3M;
	(* Controls *)
	Refresh_Auto	: BOOL:=TRUE; (* Enable automatic refresh *)
	Refresh_Now		: BOOL; 	  (* Force an immediate refresh *)
	(* Interface *)
	aPHY    : Get_ASi_PHY_Dat;
	aLCE    : Get_LCE;
	aLCEMS  : Get_LCEMS;
	aLPF	: Get_LPF;
	
END_VAR
VAR_OUTPUT
	(* Status *)
	Status_Log	: BYTE;
	Status_Vis	: DWORD;
END_VAR
VAR
	dly 	 	: TON := (PT:=T#5S);
	err 		: BYTE;
	err_old		: BYTE:=0;
END_VAR

(* Auto refresh timer *)
dly(IN:=NOT (dly.Q OR Refresh_Now OR (NOT Refresh_Auto)));
IF dly.Q THEN dly.PT:=Refresh_Period; Refresh_Now:=TRUE; END_IF

(* execute diagnostics *)
aPHY  (xExecute:=NOT Refresh_Now, enASi_Master:=SEL(ID=2,Master_1,Master_2));
aLCE  (xExecute:=NOT Refresh_Now, enASi_Master:=aPHY.enASi_Master);
aLCEMS(xExecute:=NOT Refresh_Now, enASi_Master:=aPHY.enASi_Master);
aLPF  (xExecute:=NOT Refresh_Now, enASi_Master:=aPHY.enASi_Master);
Refresh_Now:=FALSE;

(* Check status *)
IF aPHY.xReady AND aLCE.xReady AND aLCEMS.xReady AND aLPF.xReady THEN

	IF aPHY.xSE AND aPHY.xEF THEN err:=1;
	ELSIF aPHY.xPF1 THEN err:=2;
	ELSIF aPHY.xPF2 THEN err:=3;
	ELSIF aLCE.dwLCE_SA_Slaves<>0 OR aLCE.dwLCE_B_Slaves<>0 THEN err:=4;
	ELSIF aLCEMS.dwLCEMS_SA_Slaves<>0 OR aLCE.dwLCE_B_Slaves<>0 THEN err:=5;
	ELSIF aLPF.dwLPF_SA_Slaves<>0 OR aLPF.dwLPF_B_Slaves<>0 THEN err:=6;
	ELSE err:=0; END_IF

	IF err<>err_old THEN
		err_old:=err;
		CASE err OF
			0: LogEv(EL_Log,EO_ASGW,ID,1,'ASi_OK');
			1,2,3: LogEv(EL_Alarm,EO_ASGW,ID,3,'ASi_ERR');
			4,5,6: LogEv(EL_Wrn,EO_ASGW,ID,2,'ASi_SLAVE_ERR');
		END_CASE
	END_IF

	(* Log/visu status *)
	   IF err>0  AND err<4 THEN Status_Log:=2; Status_Vis:=COLOR_RED;
	ELSIF err>=4           THEN Status_Log:=1; Status_Vis:=COLOR_YELLOW;
					 	   ELSE Status_Log:=0; Status_Vis:=COLOR_GREEN;
	END_IF

END_IF

END_FUNCTION_BLOCK

// POUs/Plant_Objects/obj_PSG
FUNCTION_BLOCK obj_PSG
(* === Passage sensor ===
   v1.0[27/05/15] - Create
*)
VAR_INPUT
	(* Settings *)
	ID				: BYTE;
	POLARITY		: BOOL:=TRUE;  (* Default unoccupied polarity *)
	ERR_TIMEOUT		: TIME:=T#30M; (* Timeout for occupied barrier error *)
(*	WRN_TIMEOUT		: TIME:=T#5M;  (* Timeout fot occupied barrier warning *)*)	
(*	ACT_TIMEOUT 	: TIME:=T#7D;  (* Timeout for inactive barrier warning *)*)
(*	DISTANCE		: WORD; 	   (* Distance to 2th sensor in mm *)*)
(*  SPEED_THRESHOLD : INT;         (* Speed threshold for output trigger *)*)
	(* Ack output events *)
	SENSE_TRIG		: BOOL;
(*	SPEED_TRIG		: BOOL; *)
	(* Physical inputs *)
	PSG_IN			: BOOL;        (* Sensor input *)
(*	PSG_IN2			: BOOL;        (* Optional speed input sensor *)*)	
END_VAR
VAR_IN_OUT
	PASSAGES		: DWORD;
(*	SPEED			: AVERAGE_INT; *)	
END_VAR
VAR_OUTPUT
	SENSOR			: BOOL;
	(* Status *)
	Status_Log		: BYTE;
	Status_Vis 		: DWORD;
END_VAR
VAR
	evnt	: FLT_EVENT;
	errt	: TON;
	errtev	: FLT_EVENT;
(*	wrnt	: TON;*)
(*	actt	: TON:*)
END_VAR

SENSOR:=PSG_IN XOR POLARITY;

(* Statistics *)
evnt(IN:=SENSOR);
IF evnt.EVH THEN
	SENSE_TRIG:=TRUE;
	IF PASSAGES=16#FFFFFFFF THEN
		LogEv(EL_Wrn,EO_PSG,ID,5,'');
		PASSAGES:=1;
	ELSE
		PASSAGES:=PASSAGES+1;
	END_IF
END_IF

(* Error check *)
errt(IN:=SENSOR, PT:=ERR_TIMEOUT);
errtev(IN:=errt.Q);
IF errtev.EVH THEN
	Status_Log:=2; Status_Vis:=COLOR_RED;
	LogEv(EL_Alarm,EO_PSG,ID,2,'');
END_IF
IF errtev.EVL THEN
	Status_Log:=0; Status_Vis:=COLOR_GREEN;
	LogEv(EL_Log,EO_PSG,ID,1,'');
END_IF

ACTION StatReset:
(* Reset statistic counters *)
PASSAGES:=0;
END_ACTION

ACTION AddLogData:
//Genera la stringa di log dei passaggi	//GIURE ver 23_002

Logger.s1:=INSERT('&PSG=',WORD_TO_STRING(ID),4);
IF ID<10 THEN Logger.s1:=INSERT(Logger.s1,'0',4); END_IF

Logger.s1:=CONCAT(Logger.s1,DWORD_TO_STRING(PASSAGES));		
Logger.s1:=CONCAT(Logger.s1,';');

ADDSTRING(ADR(Logger.TData), ADR(Logger.s1), Logger.TLen);
END_ACTION

END_FUNCTION_BLOCK

// POUs/Plant_Objects/obj_ZGW
FUNCTION_BLOCK obj_ZGW
(* === ZIGBEE GATEWAY ===
   v1.0[04/06/05] - Create
*)
VAR_INPUT
	(* Settings *)
	ID				: BYTE;
	ADDRESS			: DWORD;
	Refresh_Period	: TIME:=t#3m;
	(* Controls *)
	Refresh_Auto	: BOOL:=TRUE; (* Enable automatic refresh *)
	Refresh_Now		: BOOL; 	  (* Force an immediate refresh *)
END_VAR
VAR_IN_OUT
	(* Interface *)
	MODBUS			: obj_MODBUS_TCP;
END_VAR
VAR_OUTPUT
	(* Status *)
	Status_Log		: BYTE;
	Status_Vis 		: DWORD;
END_VAR
VAR
	dly 	 	: TON := (PT:=t#5s);

	init_st		: BOOL;
	bus_st0		: BYTE;
	dev_st0		: BYTE;
END_VAR

(* Auto refresh timer *)
dly(IN:=NOT (dly.Q OR Refresh_Now OR (NOT Refresh_Auto)));
IF dly.Q THEN dly.PT:=Refresh_Period; Refresh_Now:=TRUE; END_IF
(*
(* Refresh readings *)
IF Refresh_Now THEN
	IF NOT MODBUS.MB_Lock THEN
		MODBUS.MB_Lock:=TRUE;
	END_IF
END_IF

(* Check status *)
IF NOT init_st OR MOD'ErroreSlaveModbus'<>bus_st0 OR 'ErroreSlave'<>dev_st0 THEN
	init_st:=TRUE;
	bus_st0:=M1.bError; dev_st0:=M1.utMBInfo.bMStatus;
	IF bus_st0<>0 THEN
		LogEv(EL_Alarm,EO_ZGW,ID,2,BYTE_TO_STRING(bus_st0));
		Status_Log:=2; Status_Vis:=16#2020F0;
	ELSE
		IF dev_st0<>0 THEN
			Status_Log:=2; Status_Vis:=16#2020F0;
			CASE dev_st0 OF
				000: LogEv(EL_Alarm,EO_ZGW,ID,3,'err');
				001: LogEv(EL_Wrn  ,EO_ZGW,ID,3,'wrn'); Status_Log:=1; Status_Vis:=16#20F0F0;
			ELSE
				LogEv(EL_Alarm,EO_ZGW,ID,3,BYTE_TO_STRING(dev_st0));
			END_CASE
		ELSE
			Status_Log:=0; Status_Vis:=16#20F020;
			LogEv(EL_Log,EO_ZGW,ID,1,'');
		END_IF
	END_IF
END_IF
*)

ACTION AddLogData:
Logger.s1:=INSERT('&ZGW=',BYTE_TO_STRING(ID),4);
IF ID<10 THEN Logger.s1:=INSERT(Logger.s1,'0',4); END_IF

(* NOT YET DEFINED !!! *)
Logger.s1:=CONCAT(Logger.s1,'TODEFINE');		Logger.s1:=CONCAT(Logger.s1,';');

Logger.s1:=CONCAT(Logger.s1,BYTE_TO_STRING(Status_Log));
ADDSTRING(ADR(Logger.TData), ADR(Logger.s1), Logger.TLen);
END_ACTION

END_FUNCTION_BLOCK

// POUs/WagoLibModbus_IP_01/Modbus_IP_Version
FUNCTION Modbus_IP_Version : STRING
(*Bibliotheks Version 1.12																	*)

(*Historie:1.12 new FC22 Read Mask Register implemented  								*)
(*Historie:1.11 Bugfix Master TCP 															*)
(*Historie:1.10 add documentation for  error code 16#95 									*)
(*Historie:1.9 Master TCP additional error code 16#95,xSend reset if error code<>0 		*)
(*Historie:1.8 Bugfix Master UDP 															*)
(*Historie:1.7 Bugfix Master UDP output wError												*)
(*Historie:1.6 Improvement according to FW13												*)
(*Historie:1.5 Push Bit added																	*)
(*Historie:1.4 Compiler 2.3.7.1 adaption														*)
VAR_INPUT
	xDummy:BOOL;
END_VAR
VAR
END_VAR

Modbus_IP_Version:='1.12';

END_FUNCTION

// Device/Application/VIS_CHONOEDITOR
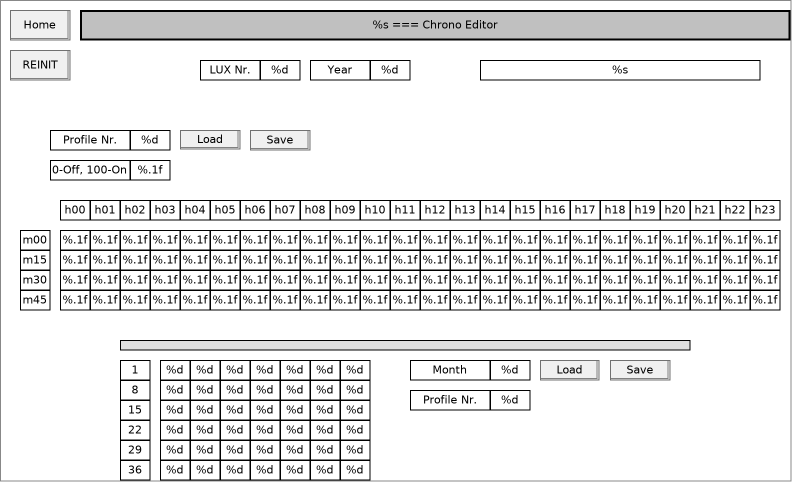
VISUALIZATION VIS_CHONOEDITOR  // 792x482
    Rectangle (200,60 60x20), "LUX Nr."
    Rectangle (260,60 40x20), "%d", text variable: CronEd.CN_Sel, colour toggle: CronEd.CN_Sel<>CronEd.CN_Act
        OnMouseDown: write the text variable via Edit, min 1, max 100, title '1'
    Rectangle (50,130 80x20), "Profile Nr."
    Rectangle (130,130 40x20), "%d", text variable: CronEd.PR_Sel, colour toggle: CronEd.PR_Sel<>CronEd.PR_Act
        OnMouseDown: write the text variable via Edit, min 1, max 10
    Rectangle (50,160 80x20), "0-Off, 100-On"
    Rectangle (130,160 40x20), "%.1f", text variable: CronEd.PR_TT
        OnMouseDown: write the text variable via Edit
    Button (180,130 60x19), "Load", pressed state: CronEd.PR_Load
        toggle CronEd.PR_Load
    Button (250,130 60x20), "Save", pressed state: CronEd.PR_Save
        toggle CronEd.PR_Save
    Rectangle (20,230 30x20), "m00"
    Rectangle (20,250 30x20), "m15"
    Rectangle (20,270 30x20), "m30"
    Rectangle (20,290 30x20), "m45"
    Rectangle (80,10 710x30), "%s === Chrono Editor", text variable: Plant_NAME
    Button (10,10 60x30), "Home"
        OnMouseUp:  Assign=PLC_VISU, Assign=PLC_VISU, Type=Assignment
    Polygon (20,210)
    RoundedRectangle (60,230 30x20), "%.1f", text variable: INT_TO_REAL(CronEd.PR.Setpoint[0])/10
        OnMouseUp: execute { CronEd.PR.Setpoint[0]:=(REAL_TO_WORD(CronEd.PR_TT*10)); }
    RoundedRectangle (60,250 30x20), "%.1f", text variable: INT_TO_REAL(CronEd.PR.Setpoint[1])/10
        OnMouseUp: execute { CronEd.PR.Setpoint[1]:=(REAL_TO_WORD(CronEd.PR_TT*10)); }
    RoundedRectangle (60,270 30x20), "%.1f", text variable: INT_TO_REAL(CronEd.PR.Setpoint[2])/10
        OnMouseUp: execute { CronEd.PR.Setpoint[2]:=(REAL_TO_WORD(CronEd.PR_TT*10)); }
    RoundedRectangle (60,290 30x20), "%.1f", text variable: INT_TO_REAL(CronEd.PR.Setpoint[3])/10
        OnMouseUp: execute { CronEd.PR.Setpoint[3]:=(REAL_TO_WORD(CronEd.PR_TT*10)); }
    Rectangle (60,200 30x20), "h00"
        OnMouseUp: execute { CronEd.PR.Setpoint[0]:=(REAL_TO_WORD(CronEd.PR_TT*10)); }
        OnMouseUp: execute { CronEd.PR.Setpoint[1]:=(REAL_TO_WORD(CronEd.PR_TT*10)); }
        OnMouseUp: execute { CronEd.PR.Setpoint[2]:=(REAL_TO_WORD(CronEd.PR_TT*10)); }
        OnMouseUp: execute { CronEd.PR.Setpoint[3]:=(REAL_TO_WORD(CronEd.PR_TT*10)); }
    RoundedRectangle (90,230 30x20), "%.1f", text variable: INT_TO_REAL(CronEd.PR.Setpoint[4])/10
        OnMouseUp: execute { CronEd.PR.Setpoint[4]:=(REAL_TO_WORD(CronEd.PR_TT*10)); }
    RoundedRectangle (90,250 30x20), "%.1f", text variable: INT_TO_REAL(CronEd.PR.Setpoint[5])/10
        OnMouseUp: execute { CronEd.PR.Setpoint[5]:=(REAL_TO_WORD(CronEd.PR_TT*10)); }
    RoundedRectangle (90,270 30x20), "%.1f", text variable: INT_TO_REAL(CronEd.PR.Setpoint[6])/10
        OnMouseUp: execute { CronEd.PR.Setpoint[6]:=(REAL_TO_WORD(CronEd.PR_TT*10)); }
    RoundedRectangle (90,290 30x20), "%.1f", text variable: INT_TO_REAL(CronEd.PR.Setpoint[7])/10
        OnMouseUp: execute { CronEd.PR.Setpoint[7]:=(REAL_TO_WORD(CronEd.PR_TT*10)); }
    Rectangle (90,200 30x20), "h01"
        OnMouseUp: execute { CronEd.PR.Setpoint[4]:=(REAL_TO_WORD(CronEd.PR_TT*10)); }
        OnMouseUp: execute { CronEd.PR.Setpoint[5]:=(REAL_TO_WORD(CronEd.PR_TT*10)); }
        OnMouseUp: execute { CronEd.PR.Setpoint[6]:=(REAL_TO_WORD(CronEd.PR_TT*10)); }
        OnMouseUp: execute { CronEd.PR.Setpoint[7]:=(REAL_TO_WORD(CronEd.PR_TT*10)); }
    RoundedRectangle (120,230 30x20), "%.1f", text variable: INT_TO_REAL(CronEd.PR.Setpoint[8])/10
        OnMouseUp: execute { CronEd.PR.Setpoint[8]:=(REAL_TO_WORD(CronEd.PR_TT*10)); }
    RoundedRectangle (120,250 30x20), "%.1f", text variable: INT_TO_REAL(CronEd.PR.Setpoint[9])/10
        OnMouseUp: execute { CronEd.PR.Setpoint[9]:=(REAL_TO_WORD(CronEd.PR_TT*10)); }
    RoundedRectangle (120,270 30x20), "%.1f", text variable: INT_TO_REAL(CronEd.PR.Setpoint[10])/10
        OnMouseUp: execute { CronEd.PR.Setpoint[10]:=(REAL_TO_WORD(CronEd.PR_TT*10)); }
    RoundedRectangle (120,290 30x20), "%.1f", text variable: INT_TO_REAL(CronEd.PR.Setpoint[11])/10
        OnMouseUp: execute { CronEd.PR.Setpoint[11]:=(REAL_TO_WORD(CronEd.PR_TT*10)); }
    Rectangle (120,200 30x20), "h02"
        OnMouseUp: execute { CronEd.PR.Setpoint[8]:=(REAL_TO_WORD(CronEd.PR_TT*10)); }
        OnMouseUp: execute { CronEd.PR.Setpoint[9]:=(REAL_TO_WORD(CronEd.PR_TT*10)); }
        OnMouseUp: execute { CronEd.PR.Setpoint[10]:=(REAL_TO_WORD(CronEd.PR_TT*10)); }
        OnMouseUp: execute { CronEd.PR.Setpoint[11]:=(REAL_TO_WORD(CronEd.PR_TT*10)); }
    RoundedRectangle (150,230 30x20), "%.1f", text variable: INT_TO_REAL(CronEd.PR.Setpoint[12])/10
        OnMouseUp: execute { CronEd.PR.Setpoint[12]:=(REAL_TO_WORD(CronEd.PR_TT*10)); }
    RoundedRectangle (150,250 30x20), "%.1f", text variable: INT_TO_REAL(CronEd.PR.Setpoint[13])/10
        OnMouseUp: execute { CronEd.PR.Setpoint[13]:=(REAL_TO_WORD(CronEd.PR_TT*10)); }
    RoundedRectangle (150,270 30x20), "%.1f", text variable: INT_TO_REAL(CronEd.PR.Setpoint[14])/10
        OnMouseUp: execute { CronEd.PR.Setpoint[14]:=(REAL_TO_WORD(CronEd.PR_TT*10)); }
    RoundedRectangle (150,290 30x20), "%.1f", text variable: INT_TO_REAL(CronEd.PR.Setpoint[15])/10
        OnMouseUp: execute { CronEd.PR.Setpoint[15]:=(REAL_TO_WORD(CronEd.PR_TT*10)); }
    Rectangle (150,200 30x20), "h03"
        OnMouseUp: execute { CronEd.PR.Setpoint[15]:=(REAL_TO_WORD(CronEd.PR_TT*10)); }
        OnMouseUp: execute { CronEd.PR.Setpoint[14]:=(REAL_TO_WORD(CronEd.PR_TT*10)); }
        OnMouseUp: execute { CronEd.PR.Setpoint[13]:=(REAL_TO_WORD(CronEd.PR_TT*10)); }
        OnMouseUp: execute { CronEd.PR.Setpoint[12]:=(REAL_TO_WORD(CronEd.PR_TT*10)); }
    RoundedRectangle (180,230 30x20), "%.1f", text variable: INT_TO_REAL(CronEd.PR.Setpoint[16])/10
        OnMouseUp: execute { CronEd.PR.Setpoint[16]:=(REAL_TO_WORD(CronEd.PR_TT*10)); }
    RoundedRectangle (180,250 30x20), "%.1f", text variable: INT_TO_REAL(CronEd.PR.Setpoint[17])/10
        OnMouseUp: execute { CronEd.PR.Setpoint[17]:=(REAL_TO_WORD(CronEd.PR_TT*10)); }
    RoundedRectangle (180,270 30x20), "%.1f", text variable: INT_TO_REAL(CronEd.PR.Setpoint[18])/10
        OnMouseUp: execute { CronEd.PR.Setpoint[18]:=(REAL_TO_WORD(CronEd.PR_TT*10)); }
    RoundedRectangle (180,290 30x20), "%.1f", text variable: INT_TO_REAL(CronEd.PR.Setpoint[19])/10
        OnMouseUp: execute { CronEd.PR.Setpoint[19]:=(REAL_TO_WORD(CronEd.PR_TT*10)); }
    Rectangle (180,200 30x20), "h04"
        OnMouseUp: execute { CronEd.PR.Setpoint[19]:=(REAL_TO_WORD(CronEd.PR_TT*10)); }
        OnMouseUp: execute { CronEd.PR.Setpoint[18]:=(REAL_TO_WORD(CronEd.PR_TT*10)); }
        OnMouseUp: execute { CronEd.PR.Setpoint[17]:=(REAL_TO_WORD(CronEd.PR_TT*10)); }
        OnMouseUp: execute { CronEd.PR.Setpoint[16]:=(REAL_TO_WORD(CronEd.PR_TT*10)); }
    RoundedRectangle (210,230 30x20), "%.1f", text variable: INT_TO_REAL(CronEd.PR.Setpoint[20])/10
        OnMouseUp: execute { CronEd.PR.Setpoint[20]:=(REAL_TO_WORD(CronEd.PR_TT*10)); }
    RoundedRectangle (210,250 30x20), "%.1f", text variable: INT_TO_REAL(CronEd.PR.Setpoint[21])/10
        OnMouseUp: execute { CronEd.PR.Setpoint[21]:=(REAL_TO_WORD(CronEd.PR_TT*10)); }
    RoundedRectangle (210,270 30x20), "%.1f", text variable: INT_TO_REAL(CronEd.PR.Setpoint[22])/10
        OnMouseUp: execute { CronEd.PR.Setpoint[22]:=(REAL_TO_WORD(CronEd.PR_TT*10)); }
    RoundedRectangle (210,290 30x20), "%.1f", text variable: INT_TO_REAL(CronEd.PR.Setpoint[23])/10
        OnMouseUp: execute { CronEd.PR.Setpoint[23]:=(REAL_TO_WORD(CronEd.PR_TT*10)); }
    Rectangle (210,200 30x20), "h05"
        OnMouseUp: execute { CronEd.PR.Setpoint[23]:=(REAL_TO_WORD(CronEd.PR_TT*10)); }
        OnMouseUp: execute { CronEd.PR.Setpoint[22]:=(REAL_TO_WORD(CronEd.PR_TT*10)); }
        OnMouseUp: execute { CronEd.PR.Setpoint[21]:=(REAL_TO_WORD(CronEd.PR_TT*10)); }
        OnMouseUp: execute { CronEd.PR.Setpoint[20]:=(REAL_TO_WORD(CronEd.PR_TT*10)); }
    RoundedRectangle (240,230 30x20), "%.1f", text variable: INT_TO_REAL(CronEd.PR.Setpoint[24])/10
        OnMouseUp: execute { CronEd.PR.Setpoint[24]:=(REAL_TO_WORD(CronEd.PR_TT*10)); }
    RoundedRectangle (240,250 30x20), "%.1f", text variable: INT_TO_REAL(CronEd.PR.Setpoint[25])/10
        OnMouseUp: execute { CronEd.PR.Setpoint[25]:=(REAL_TO_WORD(CronEd.PR_TT*10)); }
    RoundedRectangle (240,270 30x20), "%.1f", text variable: INT_TO_REAL(CronEd.PR.Setpoint[26])/10
        OnMouseUp: execute { CronEd.PR.Setpoint[26]:=(REAL_TO_WORD(CronEd.PR_TT*10)); }
    RoundedRectangle (240,290 30x20), "%.1f", text variable: INT_TO_REAL(CronEd.PR.Setpoint[27])/10
        OnMouseUp: execute { CronEd.PR.Setpoint[27]:=(REAL_TO_WORD(CronEd.PR_TT*10)); }
    Rectangle (240,200 30x20), "h06"
        OnMouseUp: execute { CronEd.PR.Setpoint[27]:=(REAL_TO_WORD(CronEd.PR_TT*10)); }
        OnMouseUp: execute { CronEd.PR.Setpoint[26]:=(REAL_TO_WORD(CronEd.PR_TT*10)); }
        OnMouseUp: execute { CronEd.PR.Setpoint[25]:=(REAL_TO_WORD(CronEd.PR_TT*10)); }
        OnMouseUp: execute { CronEd.PR.Setpoint[24]:=(REAL_TO_WORD(CronEd.PR_TT*10)); }
    RoundedRectangle (270,230 30x20), "%.1f", text variable: INT_TO_REAL(CronEd.PR.Setpoint[28])/10
        OnMouseUp: execute { CronEd.PR.Setpoint[28]:=(REAL_TO_WORD(CronEd.PR_TT*10)); }
    RoundedRectangle (270,250 30x20), "%.1f", text variable: INT_TO_REAL(CronEd.PR.Setpoint[29])/10
        OnMouseUp: execute { CronEd.PR.Setpoint[29]:=(REAL_TO_WORD(CronEd.PR_TT*10)); }
    RoundedRectangle (270,270 30x20), "%.1f", text variable: INT_TO_REAL(CronEd.PR.Setpoint[30])/10
        OnMouseUp: execute { CronEd.PR.Setpoint[30]:=(REAL_TO_WORD(CronEd.PR_TT*10)); }
    RoundedRectangle (270,290 30x20), "%.1f", text variable: INT_TO_REAL(CronEd.PR.Setpoint[31])/10
        OnMouseUp: execute { CronEd.PR.Setpoint[31]:=(REAL_TO_WORD(CronEd.PR_TT*10)); }
    Rectangle (270,200 30x20), "h07"
        OnMouseUp: execute { CronEd.PR.Setpoint[31]:=(REAL_TO_WORD(CronEd.PR_TT*10)); }
        OnMouseUp: execute { CronEd.PR.Setpoint[30]:=(REAL_TO_WORD(CronEd.PR_TT*10)); }
        OnMouseUp: execute { CronEd.PR.Setpoint[29]:=(REAL_TO_WORD(CronEd.PR_TT*10)); }
        OnMouseUp: execute { CronEd.PR.Setpoint[28]:=(REAL_TO_WORD(CronEd.PR_TT*10)); }
    RoundedRectangle (300,230 30x20), "%.1f", text variable: INT_TO_REAL(CronEd.PR.Setpoint[32])/10
        OnMouseUp: execute { CronEd.PR.Setpoint[32]:=(REAL_TO_WORD(CronEd.PR_TT*10)); }
    RoundedRectangle (300,250 30x20), "%.1f", text variable: INT_TO_REAL(CronEd.PR.Setpoint[33])/10
        OnMouseUp: execute { CronEd.PR.Setpoint[33]:=(REAL_TO_WORD(CronEd.PR_TT*10)); }
    RoundedRectangle (300,270 30x20), "%.1f", text variable: INT_TO_REAL(CronEd.PR.Setpoint[34])/10
        OnMouseUp: execute { CronEd.PR.Setpoint[34]:=(REAL_TO_WORD(CronEd.PR_TT*10)); }
    RoundedRectangle (300,290 30x20), "%.1f", text variable: INT_TO_REAL(CronEd.PR.Setpoint[35])/10
        OnMouseUp: execute { CronEd.PR.Setpoint[35]:=(REAL_TO_WORD(CronEd.PR_TT*10)); }
    Rectangle (300,200 30x20), "h08"
        OnMouseUp: execute { CronEd.PR.Setpoint[35]:=(REAL_TO_WORD(CronEd.PR_TT*10)); }
        OnMouseUp: execute { CronEd.PR.Setpoint[34]:=(REAL_TO_WORD(CronEd.PR_TT*10)); }
        OnMouseUp: execute { CronEd.PR.Setpoint[33]:=(REAL_TO_WORD(CronEd.PR_TT*10)); }
        OnMouseUp: execute { CronEd.PR.Setpoint[32]:=(REAL_TO_WORD(CronEd.PR_TT*10)); }
    RoundedRectangle (330,230 30x20), "%.1f", text variable: INT_TO_REAL(CronEd.PR.Setpoint[36])/10
        OnMouseUp: execute { CronEd.PR.Setpoint[36]:=(REAL_TO_WORD(CronEd.PR_TT*10)); }
    RoundedRectangle (330,250 30x20), "%.1f", text variable: INT_TO_REAL(CronEd.PR.Setpoint[37])/10
        OnMouseUp: execute { CronEd.PR.Setpoint[37]:=(REAL_TO_WORD(CronEd.PR_TT*10)); }
    RoundedRectangle (330,270 30x20), "%.1f", text variable: INT_TO_REAL(CronEd.PR.Setpoint[38])/10
        OnMouseUp: execute { CronEd.PR.Setpoint[38]:=(REAL_TO_WORD(CronEd.PR_TT*10)); }
    RoundedRectangle (330,290 30x20), "%.1f", text variable: INT_TO_REAL(CronEd.PR.Setpoint[39])/10
        OnMouseUp: execute { CronEd.PR.Setpoint[39]:=(REAL_TO_WORD(CronEd.PR_TT*10)); }
    Rectangle (330,200 30x20), "h09"
        OnMouseUp: execute { CronEd.PR.Setpoint[39]:=(REAL_TO_WORD(CronEd.PR_TT*10)); }
        OnMouseUp: execute { CronEd.PR.Setpoint[38]:=(REAL_TO_WORD(CronEd.PR_TT*10)); }
        OnMouseUp: execute { CronEd.PR.Setpoint[37]:=(REAL_TO_WORD(CronEd.PR_TT*10)); }
        OnMouseUp: execute { CronEd.PR.Setpoint[36]:=(REAL_TO_WORD(CronEd.PR_TT*10)); }
    RoundedRectangle (360,230 30x20), "%.1f", text variable: INT_TO_REAL(CronEd.PR.Setpoint[40])/10
        OnMouseUp: execute { CronEd.PR.Setpoint[40]:=(REAL_TO_WORD(CronEd.PR_TT*10)); }
    RoundedRectangle (360,250 30x20), "%.1f", text variable: INT_TO_REAL(CronEd.PR.Setpoint[41])/10
        OnMouseUp: execute { CronEd.PR.Setpoint[41]:=(REAL_TO_WORD(CronEd.PR_TT*10)); }
    RoundedRectangle (360,270 30x20), "%.1f", text variable: INT_TO_REAL(CronEd.PR.Setpoint[42])/10
        OnMouseUp: execute { CronEd.PR.Setpoint[42]:=(REAL_TO_WORD(CronEd.PR_TT*10)); }
    RoundedRectangle (360,290 30x20), "%.1f", text variable: INT_TO_REAL(CronEd.PR.Setpoint[43])/10
        OnMouseUp: execute { CronEd.PR.Setpoint[43]:=(REAL_TO_WORD(CronEd.PR_TT*10)); }
    Rectangle (360,200 30x20), "h10"
        OnMouseUp: execute { CronEd.PR.Setpoint[43]:=(REAL_TO_WORD(CronEd.PR_TT*10)); }
        OnMouseUp: execute { CronEd.PR.Setpoint[42]:=(REAL_TO_WORD(CronEd.PR_TT*10)); }
        OnMouseUp: execute { CronEd.PR.Setpoint[41]:=(REAL_TO_WORD(CronEd.PR_TT*10)); }
        OnMouseUp: execute { CronEd.PR.Setpoint[40]:=(REAL_TO_WORD(CronEd.PR_TT*10)); }
    RoundedRectangle (390,230 30x20), "%.1f", text variable: INT_TO_REAL(CronEd.PR.Setpoint[44])/10
        OnMouseUp: execute { CronEd.PR.Setpoint[44]:=(REAL_TO_WORD(CronEd.PR_TT*10)); }
    RoundedRectangle (390,250 30x20), "%.1f", text variable: INT_TO_REAL(CronEd.PR.Setpoint[45])/10
        OnMouseUp: execute { CronEd.PR.Setpoint[45]:=(REAL_TO_WORD(CronEd.PR_TT*10)); }
    RoundedRectangle (390,270 30x20), "%.1f", text variable: INT_TO_REAL(CronEd.PR.Setpoint[46])/10
        OnMouseUp: execute { CronEd.PR.Setpoint[46]:=(REAL_TO_WORD(CronEd.PR_TT*10)); }
    RoundedRectangle (390,290 30x20), "%.1f", text variable: INT_TO_REAL(CronEd.PR.Setpoint[47])/10
        OnMouseUp: execute { CronEd.PR.Setpoint[47]:=(REAL_TO_WORD(CronEd.PR_TT*10)); }
    Rectangle (390,200 30x20), "h11"
        OnMouseUp: execute { CronEd.PR.Setpoint[47]:=(REAL_TO_WORD(CronEd.PR_TT*10)); }
        OnMouseUp: execute { CronEd.PR.Setpoint[46]:=(REAL_TO_WORD(CronEd.PR_TT*10)); }
        OnMouseUp: execute { CronEd.PR.Setpoint[45]:=(REAL_TO_WORD(CronEd.PR_TT*10)); }
        OnMouseUp: execute { CronEd.PR.Setpoint[44]:=(REAL_TO_WORD(CronEd.PR_TT*10)); }
    RoundedRectangle (420,230 30x20), "%.1f", text variable: INT_TO_REAL(CronEd.PR.Setpoint[48])/10
        OnMouseUp: execute { CronEd.PR.Setpoint[48]:=(REAL_TO_WORD(CronEd.PR_TT*10)); }
    RoundedRectangle (420,250 30x20), "%.1f", text variable: INT_TO_REAL(CronEd.PR.Setpoint[49])/10
        OnMouseUp: execute { CronEd.PR.Setpoint[49]:=(REAL_TO_WORD(CronEd.PR_TT*10)); }
    RoundedRectangle (420,270 30x20), "%.1f", text variable: INT_TO_REAL(CronEd.PR.Setpoint[50])/10
        OnMouseUp: execute { CronEd.PR.Setpoint[50]:=(REAL_TO_WORD(CronEd.PR_TT*10)); }
    RoundedRectangle (420,290 30x20), "%.1f", text variable: INT_TO_REAL(CronEd.PR.Setpoint[51])/10
        OnMouseUp: execute { CronEd.PR.Setpoint[51]:=(REAL_TO_WORD(CronEd.PR_TT*10)); }
    Rectangle (420,200 30x20), "h12"
        OnMouseUp: execute { CronEd.PR.Setpoint[51]:=(REAL_TO_WORD(CronEd.PR_TT*10)); }
        OnMouseUp: execute { CronEd.PR.Setpoint[50]:=(REAL_TO_WORD(CronEd.PR_TT*10)); }
        OnMouseUp: execute { CronEd.PR.Setpoint[49]:=(REAL_TO_WORD(CronEd.PR_TT*10)); }
        OnMouseUp: execute { CronEd.PR.Setpoint[48]:=(REAL_TO_WORD(CronEd.PR_TT*10)); }
    RoundedRectangle (450,230 30x20), "%.1f", text variable: INT_TO_REAL(CronEd.PR.Setpoint[52])/10
        OnMouseUp: execute { CronEd.PR.Setpoint[52]:=(REAL_TO_WORD(CronEd.PR_TT*10)); }
    RoundedRectangle (450,250 30x20), "%.1f", text variable: INT_TO_REAL(CronEd.PR.Setpoint[53])/10
        OnMouseUp: execute { CronEd.PR.Setpoint[53]:=(REAL_TO_WORD(CronEd.PR_TT*10)); }
    RoundedRectangle (450,270 30x20), "%.1f", text variable: INT_TO_REAL(CronEd.PR.Setpoint[54])/10
        OnMouseUp: execute { CronEd.PR.Setpoint[54]:=(REAL_TO_WORD(CronEd.PR_TT*10)); }
    RoundedRectangle (450,290 30x20), "%.1f", text variable: INT_TO_REAL(CronEd.PR.Setpoint[55])/10
        OnMouseUp: execute { CronEd.PR.Setpoint[55]:=(REAL_TO_WORD(CronEd.PR_TT*10)); }
    Rectangle (450,200 30x20), "h13"
        OnMouseUp: execute { CronEd.PR.Setpoint[55]:=(REAL_TO_WORD(CronEd.PR_TT*10)); }
        OnMouseUp: execute { CronEd.PR.Setpoint[54]:=(REAL_TO_WORD(CronEd.PR_TT*10)); }
        OnMouseUp: execute { CronEd.PR.Setpoint[53]:=(REAL_TO_WORD(CronEd.PR_TT*10)); }
        OnMouseUp: execute { CronEd.PR.Setpoint[52]:=(REAL_TO_WORD(CronEd.PR_TT*10)); }
    RoundedRectangle (480,230 30x20), "%.1f", text variable: INT_TO_REAL(CronEd.PR.Setpoint[56])/10
        OnMouseUp: execute { CronEd.PR.Setpoint[56]:=(REAL_TO_WORD(CronEd.PR_TT*10)); }
    RoundedRectangle (480,250 30x20), "%.1f", text variable: INT_TO_REAL(CronEd.PR.Setpoint[57])/10
        OnMouseUp: execute { CronEd.PR.Setpoint[57]:=(REAL_TO_WORD(CronEd.PR_TT*10)); }
    RoundedRectangle (480,270 30x20), "%.1f", text variable: INT_TO_REAL(CronEd.PR.Setpoint[58])/10
        OnMouseUp: execute { CronEd.PR.Setpoint[58]:=(REAL_TO_WORD(CronEd.PR_TT*10)); }
    RoundedRectangle (480,290 30x20), "%.1f", text variable: INT_TO_REAL(CronEd.PR.Setpoint[59])/10
        OnMouseUp: execute { CronEd.PR.Setpoint[59]:=(REAL_TO_WORD(CronEd.PR_TT*10)); }
    Rectangle (480,200 30x20), "h14"
        OnMouseUp: execute { CronEd.PR.Setpoint[59]:=(REAL_TO_WORD(CronEd.PR_TT*10)); }
        OnMouseUp: execute { CronEd.PR.Setpoint[58]:=(REAL_TO_WORD(CronEd.PR_TT*10)); }
        OnMouseUp: execute { CronEd.PR.Setpoint[57]:=(REAL_TO_WORD(CronEd.PR_TT*10)); }
        OnMouseUp: execute { CronEd.PR.Setpoint[56]:=(REAL_TO_WORD(CronEd.PR_TT*10)); }
    RoundedRectangle (510,230 30x20), "%.1f", text variable: INT_TO_REAL(CronEd.PR.Setpoint[60])/10
        OnMouseUp: execute { CronEd.PR.Setpoint[60]:=(REAL_TO_WORD(CronEd.PR_TT*10)); }
    RoundedRectangle (510,250 30x20), "%.1f", text variable: INT_TO_REAL(CronEd.PR.Setpoint[61])/10
        OnMouseUp: execute { CronEd.PR.Setpoint[61]:=(REAL_TO_WORD(CronEd.PR_TT*10)); }
    RoundedRectangle (510,270 30x20), "%.1f", text variable: INT_TO_REAL(CronEd.PR.Setpoint[62])/10
        OnMouseUp: execute { CronEd.PR.Setpoint[62]:=(REAL_TO_WORD(CronEd.PR_TT*10)); }
    RoundedRectangle (510,290 30x20), "%.1f", text variable: INT_TO_REAL(CronEd.PR.Setpoint[63])/10
        OnMouseUp: execute { CronEd.PR.Setpoint[63]:=(REAL_TO_WORD(CronEd.PR_TT*10)); }
    Rectangle (510,200 30x20), "h15"
        OnMouseUp: execute { CronEd.PR.Setpoint[63]:=(REAL_TO_WORD(CronEd.PR_TT*10)); }
        OnMouseUp: execute { CronEd.PR.Setpoint[62]:=(REAL_TO_WORD(CronEd.PR_TT*10)); }
        OnMouseUp: execute { CronEd.PR.Setpoint[61]:=(REAL_TO_WORD(CronEd.PR_TT*10)); }
        OnMouseUp: execute { CronEd.PR.Setpoint[60]:=(REAL_TO_WORD(CronEd.PR_TT*10)); }
    RoundedRectangle (540,230 30x20), "%.1f", text variable: INT_TO_REAL(CronEd.PR.Setpoint[64])/10
        OnMouseUp: execute { CronEd.PR.Setpoint[64]:=(REAL_TO_WORD(CronEd.PR_TT*10)); }
    RoundedRectangle (540,250 30x20), "%.1f", text variable: INT_TO_REAL(CronEd.PR.Setpoint[65])/10
        OnMouseUp: execute { CronEd.PR.Setpoint[65]:=(REAL_TO_WORD(CronEd.PR_TT*10)); }
    RoundedRectangle (540,270 30x20), "%.1f", text variable: INT_TO_REAL(CronEd.PR.Setpoint[66])/10
        OnMouseUp: execute { CronEd.PR.Setpoint[66]:=(REAL_TO_WORD(CronEd.PR_TT*10)); }
    RoundedRectangle (540,290 30x20), "%.1f", text variable: INT_TO_REAL(CronEd.PR.Setpoint[67])/10
        OnMouseUp: execute { CronEd.PR.Setpoint[67]:=(REAL_TO_WORD(CronEd.PR_TT*10)); }
    Rectangle (540,200 30x20), "h16"
        OnMouseUp: execute { CronEd.PR.Setpoint[67]:=(REAL_TO_WORD(CronEd.PR_TT*10)); }
        OnMouseUp: execute { CronEd.PR.Setpoint[66]:=(REAL_TO_WORD(CronEd.PR_TT*10)); }
        OnMouseUp: execute { CronEd.PR.Setpoint[65]:=(REAL_TO_WORD(CronEd.PR_TT*10)); }
        OnMouseUp: execute { CronEd.PR.Setpoint[64]:=(REAL_TO_WORD(CronEd.PR_TT*10)); }
    RoundedRectangle (570,230 30x20), "%.1f", text variable: INT_TO_REAL(CronEd.PR.Setpoint[68])/10
        OnMouseUp: execute { CronEd.PR.Setpoint[68]:=(REAL_TO_WORD(CronEd.PR_TT*10)); }
    RoundedRectangle (570,250 30x20), "%.1f", text variable: INT_TO_REAL(CronEd.PR.Setpoint[69])/10
        OnMouseUp: execute { CronEd.PR.Setpoint[69]:=(REAL_TO_WORD(CronEd.PR_TT*10)); }
    RoundedRectangle (570,270 30x20), "%.1f", text variable: INT_TO_REAL(CronEd.PR.Setpoint[70])/10
        OnMouseUp: execute { CronEd.PR.Setpoint[70]:=(REAL_TO_WORD(CronEd.PR_TT*10)); }
    RoundedRectangle (570,290 30x20), "%.1f", text variable: INT_TO_REAL(CronEd.PR.Setpoint[71])/10
        OnMouseUp: execute { CronEd.PR.Setpoint[71]:=(REAL_TO_WORD(CronEd.PR_TT*10)); }
    Rectangle (570,200 30x20), "h17"
        OnMouseUp: execute { CronEd.PR.Setpoint[71]:=(REAL_TO_WORD(CronEd.PR_TT*10)); }
        OnMouseUp: execute { CronEd.PR.Setpoint[70]:=(REAL_TO_WORD(CronEd.PR_TT*10)); }
        OnMouseUp: execute { CronEd.PR.Setpoint[69]:=(REAL_TO_WORD(CronEd.PR_TT*10)); }
        OnMouseUp: execute { CronEd.PR.Setpoint[68]:=(REAL_TO_WORD(CronEd.PR_TT*10)); }
    RoundedRectangle (600,230 30x20), "%.1f", text variable: INT_TO_REAL(CronEd.PR.Setpoint[72])/10
        OnMouseUp: execute { CronEd.PR.Setpoint[72]:=(REAL_TO_WORD(CronEd.PR_TT*10)); }
    RoundedRectangle (600,250 30x20), "%.1f", text variable: INT_TO_REAL(CronEd.PR.Setpoint[73])/10
        OnMouseUp: execute { CronEd.PR.Setpoint[73]:=(REAL_TO_WORD(CronEd.PR_TT*10)); }
    RoundedRectangle (600,270 30x20), "%.1f", text variable: INT_TO_REAL(CronEd.PR.Setpoint[74])/10
        OnMouseUp: execute { CronEd.PR.Setpoint[74]:=(REAL_TO_WORD(CronEd.PR_TT*10)); }
    RoundedRectangle (600,290 30x20), "%.1f", text variable: INT_TO_REAL(CronEd.PR.Setpoint[75])/10
        OnMouseUp: execute { CronEd.PR.Setpoint[75]:=(REAL_TO_WORD(CronEd.PR_TT*10)); }
    Rectangle (600,200 30x20), "h18"
        OnMouseUp: execute { CronEd.PR.Setpoint[75]:=(REAL_TO_WORD(CronEd.PR_TT*10)); }
        OnMouseUp: execute { CronEd.PR.Setpoint[74]:=(REAL_TO_WORD(CronEd.PR_TT*10)); }
        OnMouseUp: execute { CronEd.PR.Setpoint[73]:=(REAL_TO_WORD(CronEd.PR_TT*10)); }
        OnMouseUp: execute { CronEd.PR.Setpoint[72]:=(REAL_TO_WORD(CronEd.PR_TT*10)); }
    RoundedRectangle (630,230 30x20), "%.1f", text variable: INT_TO_REAL(CronEd.PR.Setpoint[76])/10
        OnMouseUp: execute { CronEd.PR.Setpoint[76]:=(REAL_TO_WORD(CronEd.PR_TT*10)); }
    RoundedRectangle (630,250 30x20), "%.1f", text variable: INT_TO_REAL(CronEd.PR.Setpoint[77])/10
        OnMouseUp: execute { CronEd.PR.Setpoint[77]:=(REAL_TO_WORD(CronEd.PR_TT*10)); }
    RoundedRectangle (630,270 30x20), "%.1f", text variable: INT_TO_REAL(CronEd.PR.Setpoint[78])/10
        OnMouseUp: execute { CronEd.PR.Setpoint[78]:=(REAL_TO_WORD(CronEd.PR_TT*10)); }
    RoundedRectangle (630,290 30x20), "%.1f", text variable: INT_TO_REAL(CronEd.PR.Setpoint[79])/10
        OnMouseUp: execute { CronEd.PR.Setpoint[79]:=(REAL_TO_WORD(CronEd.PR_TT*10)); }
    Rectangle (630,200 30x20), "h19"
        OnMouseUp: execute { CronEd.PR.Setpoint[79]:=(REAL_TO_WORD(CronEd.PR_TT*10)); }
        OnMouseUp: execute { CronEd.PR.Setpoint[78]:=(REAL_TO_WORD(CronEd.PR_TT*10)); }
        OnMouseUp: execute { CronEd.PR.Setpoint[77]:=(REAL_TO_WORD(CronEd.PR_TT*10)); }
        OnMouseUp: execute { CronEd.PR.Setpoint[76]:=(REAL_TO_WORD(CronEd.PR_TT*10)); }
    RoundedRectangle (660,230 30x20), "%.1f", text variable: INT_TO_REAL(CronEd.PR.Setpoint[80])/10
        OnMouseUp: execute { CronEd.PR.Setpoint[80]:=(REAL_TO_WORD(CronEd.PR_TT*10)); }
    RoundedRectangle (660,250 30x20), "%.1f", text variable: INT_TO_REAL(CronEd.PR.Setpoint[81])/10
        OnMouseUp: execute { CronEd.PR.Setpoint[81]:=(REAL_TO_WORD(CronEd.PR_TT*10)); }
    RoundedRectangle (660,270 30x20), "%.1f", text variable: INT_TO_REAL(CronEd.PR.Setpoint[82])/10
        OnMouseUp: execute { CronEd.PR.Setpoint[82]:=(REAL_TO_WORD(CronEd.PR_TT*10)); }
    RoundedRectangle (660,290 30x20), "%.1f", text variable: INT_TO_REAL(CronEd.PR.Setpoint[83])/10
        OnMouseUp: execute { CronEd.PR.Setpoint[83]:=(REAL_TO_WORD(CronEd.PR_TT*10)); }
    Rectangle (660,200 30x20), "h20"
        OnMouseUp: execute { CronEd.PR.Setpoint[83]:=(REAL_TO_WORD(CronEd.PR_TT*10)); }
        OnMouseUp: execute { CronEd.PR.Setpoint[82]:=(REAL_TO_WORD(CronEd.PR_TT*10)); }
        OnMouseUp: execute { CronEd.PR.Setpoint[81]:=(REAL_TO_WORD(CronEd.PR_TT*10)); }
        OnMouseUp: execute { CronEd.PR.Setpoint[80]:=(REAL_TO_WORD(CronEd.PR_TT*10)); }
    RoundedRectangle (690,230 30x20), "%.1f", text variable: INT_TO_REAL(CronEd.PR.Setpoint[84])/10
        OnMouseUp: execute { CronEd.PR.Setpoint[84]:=(REAL_TO_WORD(CronEd.PR_TT*10)); }
    RoundedRectangle (690,250 30x20), "%.1f", text variable: INT_TO_REAL(CronEd.PR.Setpoint[85])/10
        OnMouseUp: execute { CronEd.PR.Setpoint[85]:=(REAL_TO_WORD(CronEd.PR_TT*10)); }
    RoundedRectangle (690,270 30x20), "%.1f", text variable: INT_TO_REAL(CronEd.PR.Setpoint[86])/10
        OnMouseUp: execute { CronEd.PR.Setpoint[86]:=(REAL_TO_WORD(CronEd.PR_TT*10)); }
    RoundedRectangle (690,290 30x20), "%.1f", text variable: INT_TO_REAL(CronEd.PR.Setpoint[87])/10
        OnMouseUp: execute { CronEd.PR.Setpoint[87]:=(REAL_TO_WORD(CronEd.PR_TT*10)); }
    Rectangle (690,200 30x20), "h21"
        OnMouseUp: execute { CronEd.PR.Setpoint[87]:=(REAL_TO_WORD(CronEd.PR_TT*10)); }
        OnMouseUp: execute { CronEd.PR.Setpoint[86]:=(REAL_TO_WORD(CronEd.PR_TT*10)); }
        OnMouseUp: execute { CronEd.PR.Setpoint[85]:=(REAL_TO_WORD(CronEd.PR_TT*10)); }
        OnMouseUp: execute { CronEd.PR.Setpoint[84]:=(REAL_TO_WORD(CronEd.PR_TT*10)); }
    RoundedRectangle (720,230 30x20), "%.1f", text variable: INT_TO_REAL(CronEd.PR.Setpoint[88])/10
        OnMouseUp: execute { CronEd.PR.Setpoint[88]:=(REAL_TO_WORD(CronEd.PR_TT*10)); }
    RoundedRectangle (720,250 30x20), "%.1f", text variable: INT_TO_REAL(CronEd.PR.Setpoint[89])/10
        OnMouseUp: execute { CronEd.PR.Setpoint[89]:=(REAL_TO_WORD(CronEd.PR_TT*10)); }
    RoundedRectangle (720,270 30x20), "%.1f", text variable: INT_TO_REAL(CronEd.PR.Setpoint[90])/10
        OnMouseUp: execute { CronEd.PR.Setpoint[90]:=(REAL_TO_WORD(CronEd.PR_TT*10)); }
    RoundedRectangle (720,290 30x20), "%.1f", text variable: INT_TO_REAL(CronEd.PR.Setpoint[91])/10
        OnMouseUp: execute { CronEd.PR.Setpoint[91]:=(REAL_TO_WORD(CronEd.PR_TT*10)); }
    Rectangle (720,200 30x20), "h22"
        OnMouseUp: execute { CronEd.PR.Setpoint[91]:=(REAL_TO_WORD(CronEd.PR_TT*10)); }
        OnMouseUp: execute { CronEd.PR.Setpoint[90]:=(REAL_TO_WORD(CronEd.PR_TT*10)); }
        OnMouseUp: execute { CronEd.PR.Setpoint[89]:=(REAL_TO_WORD(CronEd.PR_TT*10)); }
        OnMouseUp: execute { CronEd.PR.Setpoint[88]:=(REAL_TO_WORD(CronEd.PR_TT*10)); }
    RoundedRectangle (750,230 30x20), "%.1f", text variable: INT_TO_REAL(CronEd.PR.Setpoint[92])/10
        OnMouseUp: execute { CronEd.PR.Setpoint[92]:=(REAL_TO_WORD(CronEd.PR_TT*10)); }
    RoundedRectangle (750,250 30x20), "%.1f", text variable: INT_TO_REAL(CronEd.PR.Setpoint[93])/10
        OnMouseUp: execute { CronEd.PR.Setpoint[93]:=(REAL_TO_WORD(CronEd.PR_TT*10)); }
    RoundedRectangle (750,270 30x20), "%.1f", text variable: INT_TO_REAL(CronEd.PR.Setpoint[94])/10
        OnMouseUp: execute { CronEd.PR.Setpoint[94]:=(REAL_TO_WORD(CronEd.PR_TT*10)); }
    RoundedRectangle (750,290 30x20), "%.1f", text variable: INT_TO_REAL(CronEd.PR.Setpoint[95])/10
        OnMouseUp: execute { CronEd.PR.Setpoint[95]:=(REAL_TO_WORD(CronEd.PR_TT*10)); }
    Rectangle (750,200 30x20), "h23"
        OnMouseUp: execute { CronEd.PR.Setpoint[95]:=(REAL_TO_WORD(CronEd.PR_TT*10)); }
        OnMouseUp: execute { CronEd.PR.Setpoint[94]:=(REAL_TO_WORD(CronEd.PR_TT*10)); }
        OnMouseUp: execute { CronEd.PR.Setpoint[93]:=(REAL_TO_WORD(CronEd.PR_TT*10)); }
        OnMouseUp: execute { CronEd.PR.Setpoint[92]:=(REAL_TO_WORD(CronEd.PR_TT*10)); }
    Rectangle (410,360 80x20), "Month"
    Rectangle (490,360 40x20), "%d", text variable: CronEd.CA_Sel, colour toggle: CronEd.CA_Sel<>CronEd.CA_Act
        OnMouseDown: write the text variable via Edit, min 1, max 12
    Rectangle (410,390 80x20), "Profile Nr."
    Rectangle (490,390 40x20), "%d", text variable: CronEd.CA_TPR
        OnMouseDown: write the text variable via Edit, min 0, max 10
    Button (540,360 59x20), "Load", pressed state: CronEd.CA_Load
        toggle CronEd.CA_Load
    Button (610,360 60x20), "Save", pressed state: CronEd.CA_Save
        toggle CronEd.CA_Save
    RoundedRectangle (160,360 30x20), "%d", text variable: CronEd.CA.Profile[0], colour toggle: CronEd.CA.Profile[0]=0, invisible if: CronEd.CA_DayF>0
        OnMouseUp: execute { CronEd.CA.Profile[0]:=(CronEd.CA_TPR); }
    Rectangle (120,360 30x20), "1"
    RoundedRectangle (190,360 30x20), "%d", text variable: CronEd.CA.Profile[1], colour toggle: CronEd.CA.Profile[1]=0, invisible if: CronEd.CA_DayF>1
        OnMouseUp: execute { CronEd.CA.Profile[1]:=(CronEd.CA_TPR); }
    RoundedRectangle (220,360 30x20), "%d", text variable: CronEd.CA.Profile[2], colour toggle: CronEd.CA.Profile[2]=0, invisible if: CronEd.CA_DayF>2
        OnMouseUp: execute { CronEd.CA.Profile[2]:=(CronEd.CA_TPR); }
    RoundedRectangle (250,360 30x20), "%d", text variable: CronEd.CA.Profile[3], colour toggle: CronEd.CA.Profile[3]=0, invisible if: CronEd.CA_DayF>3
        OnMouseUp: execute { CronEd.CA.Profile[3]:=(CronEd.CA_TPR); }
    RoundedRectangle (280,360 30x20), "%d", text variable: CronEd.CA.Profile[4], colour toggle: CronEd.CA.Profile[4]=0, invisible if: CronEd.CA_DayF>4
        OnMouseUp: execute { CronEd.CA.Profile[4]:=(CronEd.CA_TPR); }
    RoundedRectangle (310,360 30x20), "%d", text variable: CronEd.CA.Profile[5], colour toggle: CronEd.CA.Profile[5]=0, invisible if: CronEd.CA_DayF>5
        OnMouseUp: execute { CronEd.CA.Profile[5]:=(CronEd.CA_TPR); }
    RoundedRectangle (340,360 30x20), "%d", text variable: CronEd.CA.Profile[6], colour toggle: CronEd.CA.Profile[6]=0
        OnMouseUp: execute { CronEd.CA.Profile[6]:=(CronEd.CA_TPR); }
    RoundedRectangle (160,380 30x20), "%d", text variable: CronEd.CA.Profile[7], colour toggle: CronEd.CA.Profile[7]=0
        OnMouseUp: execute { CronEd.CA.Profile[7]:=(CronEd.CA_TPR); }
    Rectangle (120,380 30x20), "8"
    RoundedRectangle (190,380 30x20), "%d", text variable: CronEd.CA.Profile[8], colour toggle: CronEd.CA.Profile[8]=0
        OnMouseUp: execute { CronEd.CA.Profile[8]:=(CronEd.CA_TPR); }
    RoundedRectangle (220,380 30x20), "%d", text variable: CronEd.CA.Profile[9], colour toggle: CronEd.CA.Profile[9]=0
        OnMouseUp: execute { CronEd.CA.Profile[9]:=(CronEd.CA_TPR); }
    RoundedRectangle (250,380 30x20), "%d", text variable: CronEd.CA.Profile[10], colour toggle: CronEd.CA.Profile[10]=0
        OnMouseUp: execute { CronEd.CA.Profile[10]:=(CronEd.CA_TPR); }
    RoundedRectangle (280,380 30x20), "%d", text variable: CronEd.CA.Profile[11], colour toggle: CronEd.CA.Profile[11]=0
        OnMouseUp: execute { CronEd.CA.Profile[11]:=(CronEd.CA_TPR); }
    RoundedRectangle (310,380 30x20), "%d", text variable: CronEd.CA.Profile[12], colour toggle: CronEd.CA.Profile[12]=0
        OnMouseUp: execute { CronEd.CA.Profile[12]:=(CronEd.CA_TPR); }
    RoundedRectangle (340,380 30x20), "%d", text variable: CronEd.CA.Profile[13], colour toggle: CronEd.CA.Profile[13]=0
        OnMouseUp: execute { CronEd.CA.Profile[13]:=(CronEd.CA_TPR); }
    RoundedRectangle (160,400 30x20), "%d", text variable: CronEd.CA.Profile[14], colour toggle: CronEd.CA.Profile[14]=0
        OnMouseUp: execute { CronEd.CA.Profile[14]:=(CronEd.CA_TPR); }
    Rectangle (120,400 30x20), "15"
    RoundedRectangle (190,400 30x20), "%d", text variable: CronEd.CA.Profile[15], colour toggle: CronEd.CA.Profile[15]=0
        OnMouseUp: execute { CronEd.CA.Profile[15]:=(CronEd.CA_TPR); }
    RoundedRectangle (220,400 30x20), "%d", text variable: CronEd.CA.Profile[16], colour toggle: CronEd.CA.Profile[16]=0
        OnMouseUp: execute { CronEd.CA.Profile[16]:=(CronEd.CA_TPR); }
    RoundedRectangle (250,400 30x20), "%d", text variable: CronEd.CA.Profile[17], colour toggle: CronEd.CA.Profile[17]=0
        OnMouseUp: execute { CronEd.CA.Profile[17]:=(CronEd.CA_TPR); }
    RoundedRectangle (280,400 30x20), "%d", text variable: CronEd.CA.Profile[18], colour toggle: CronEd.CA.Profile[18]=0
        OnMouseUp: execute { CronEd.CA.Profile[18]:=(CronEd.CA_TPR); }
    RoundedRectangle (310,400 30x20), "%d", text variable: CronEd.CA.Profile[19], colour toggle: CronEd.CA.Profile[19]=0
        OnMouseUp: execute { CronEd.CA.Profile[19]:=(CronEd.CA_TPR); }
    RoundedRectangle (340,400 30x20), "%d", text variable: CronEd.CA.Profile[20], colour toggle: CronEd.CA.Profile[20]=0
        OnMouseUp: execute { CronEd.CA.Profile[20]:=(CronEd.CA_TPR); }
    RoundedRectangle (160,420 30x20), "%d", text variable: CronEd.CA.Profile[21], colour toggle: CronEd.CA.Profile[21]=0
        OnMouseUp: execute { CronEd.CA.Profile[21]:=(CronEd.CA_TPR); }
    Rectangle (120,420 30x20), "22"
    RoundedRectangle (190,420 30x20), "%d", text variable: CronEd.CA.Profile[22], colour toggle: CronEd.CA.Profile[22]=0
        OnMouseUp: execute { CronEd.CA.Profile[22]:=(CronEd.CA_TPR); }
    RoundedRectangle (220,420 30x20), "%d", text variable: CronEd.CA.Profile[23], colour toggle: CronEd.CA.Profile[23]=0
        OnMouseUp: execute { CronEd.CA.Profile[23]:=(CronEd.CA_TPR); }
    RoundedRectangle (250,420 30x20), "%d", text variable: CronEd.CA.Profile[24], colour toggle: CronEd.CA.Profile[24]=0
        OnMouseUp: execute { CronEd.CA.Profile[24]:=(CronEd.CA_TPR); }
    RoundedRectangle (280,420 30x20), "%d", text variable: CronEd.CA.Profile[25], colour toggle: CronEd.CA.Profile[25]=0
        OnMouseUp: execute { CronEd.CA.Profile[25]:=(CronEd.CA_TPR); }
    RoundedRectangle (310,420 30x20), "%d", text variable: CronEd.CA.Profile[26], colour toggle: CronEd.CA.Profile[26]=0
        OnMouseUp: execute { CronEd.CA.Profile[26]:=(CronEd.CA_TPR); }
    RoundedRectangle (340,420 30x20), "%d", text variable: CronEd.CA.Profile[27], colour toggle: CronEd.CA.Profile[27]=0
        OnMouseUp: execute { CronEd.CA.Profile[27]:=(CronEd.CA_TPR); }
    RoundedRectangle (160,440 30x20), "%d", text variable: CronEd.CA.Profile[28], colour toggle: CronEd.CA.Profile[28]=0
        OnMouseUp: execute { CronEd.CA.Profile[28]:=(CronEd.CA_TPR); }
    Rectangle (120,440 30x20), "29"
    RoundedRectangle (190,440 30x20), "%d", text variable: CronEd.CA.Profile[29], colour toggle: CronEd.CA.Profile[29]=0
        OnMouseUp: execute { CronEd.CA.Profile[29]:=(CronEd.CA_TPR); }
    RoundedRectangle (220,440 30x20), "%d", text variable: CronEd.CA.Profile[30], colour toggle: CronEd.CA.Profile[30]=0
        OnMouseUp: execute { CronEd.CA.Profile[30]:=(CronEd.CA_TPR); }
    RoundedRectangle (250,440 30x20), "%d", text variable: CronEd.CA.Profile[31], colour toggle: CronEd.CA.Profile[31]=0
        OnMouseUp: execute { CronEd.CA.Profile[31]:=(CronEd.CA_TPR); }
    RoundedRectangle (280,440 30x20), "%d", text variable: CronEd.CA.Profile[32], colour toggle: CronEd.CA.Profile[32]=0, invisible if: CronEd.CA_DayL<32
        OnMouseUp: execute { CronEd.CA.Profile[32]:=(CronEd.CA_TPR); }
    RoundedRectangle (310,440 30x20), "%d", text variable: CronEd.CA.Profile[33], colour toggle: CronEd.CA.Profile[33]=0, invisible if: CronEd.CA_DayL<33
        OnMouseUp: execute { CronEd.CA.Profile[33]:=(CronEd.CA_TPR); }
    RoundedRectangle (340,440 30x20), "%d", text variable: CronEd.CA.Profile[34], colour toggle: CronEd.CA.Profile[34]=0, invisible if: CronEd.CA_DayL<34
        OnMouseUp: execute { CronEd.CA.Profile[34]:=(CronEd.CA_TPR); }
    RoundedRectangle (160,460 30x20), "%d", text variable: CronEd.CA.Profile[35], colour toggle: CronEd.CA.Profile[35]=0, invisible if: CronEd.CA_DayL<35
        OnMouseUp: execute { CronEd.CA.Profile[35]:=(CronEd.CA_TPR); }
    Rectangle (120,460 30x20), "36", invisible if: CronEd.CA_DayL<35
    RoundedRectangle (190,460 30x20), "%d", text variable: CronEd.CA.Profile[36], colour toggle: CronEd.CA.Profile[36]=0, invisible if: CronEd.CA_DayL<36
        OnMouseUp: execute { CronEd.CA.Profile[36]:=(CronEd.CA_TPR); }
    RoundedRectangle (220,460 30x20), "%d", text variable: CronEd.CA.Profile[37], colour toggle: CronEd.CA.Profile[37]=0, invisible if: CronEd.CA_DayL<37
        OnMouseUp: execute { CronEd.CA.Profile[37]:=(CronEd.CA_TPR); }
    RoundedRectangle (250,460 30x20), "%d", text variable: CronEd.CA.Profile[38], colour toggle: CronEd.CA.Profile[38]=0, invisible if: CronEd.CA_DayL<38
        OnMouseUp: execute { CronEd.CA.Profile[38]:=(CronEd.CA_TPR); }
    RoundedRectangle (280,460 30x20), "%d", text variable: CronEd.CA.Profile[39], colour toggle: CronEd.CA.Profile[39]=0, invisible if: CronEd.CA_DayL<39
        OnMouseUp: execute { CronEd.CA.Profile[39]:=(CronEd.CA_TPR); }
    RoundedRectangle (310,460 30x20), "%d", text variable: CronEd.CA.Profile[40], colour toggle: CronEd.CA.Profile[40]=0, invisible if: CronEd.CA_DayL<40
        OnMouseUp: execute { CronEd.CA.Profile[40]:=(CronEd.CA_TPR); }
    RoundedRectangle (340,460 30x20), "%d", text variable: CronEd.CA.Profile[41], colour toggle: CronEd.CA.Profile[41]=0, invisible if: CronEd.CA_DayL<41
        OnMouseUp: execute { CronEd.CA.Profile[41]:=(CronEd.CA_TPR); }
    Rectangle (310,60 60x20), "Year"
    Rectangle (370,60 40x20), "%d", text variable: CronEd.CN_YSel, colour toggle: CronEd.CN_YSel<>CronEd.CN_YAct
        OnMouseDown: write the text variable via Edit, min 2000, max 2100, title '1'
    Rectangle (120,340 570x10)
    Rectangle (480,60 280x20), "%s", text variable: CronEd.Message
    Button (10,50 60x30), "REINIT"
        OnMouseClick: execute {
            CRON[1].InitOK:=(FALSE);
            CRON[2].InitOK:=(FALSE);
            CRON[3].InitOK:=(FALSE);
            CRON[4].InitOK:=(FALSE);
            CRON[5].InitOK:=(FALSE);
            CRON[6].InitOK:=(FALSE);
            CRON[7].InitOK:=(FALSE);
            CRON[8].InitOK:=(FALSE);
            CRON[9].InitOK:=(FALSE);
            CRON[10].InitOK:=(FALSE);
            CRON[11].InitOK:=(FALSE);
            CRON[12].InitOK:=(FALSE);
            CRON[13].InitOK:=(FALSE);
            CRON[14].InitOK:=(FALSE);
            CRON[15].InitOK:=(FALSE);
            CRON[16].InitOK:=(FALSE);
            CRON[17].InitOK:=(FALSE);
            CRON[18].InitOK:=(FALSE);
            CRON[19].InitOK:=(FALSE);
            CRON[20].InitOK:=(FALSE);
            CRON[21].InitOK:=(FALSE);
            CRON[22].InitOK:=(FALSE);
            CRON[23].InitOK:=(FALSE);
            CRON[24].InitOK:=(FALSE);
            CRON[25].InitOK:=(FALSE);
            CRON[26].InitOK:=(FALSE);
            CRON[27].InitOK:=(FALSE);
            CRON[28].InitOK:=(FALSE);
            CRON[29].InitOK:=(FALSE);
            CRON[30].InitOK:=(FALSE);
            CRON[31].InitOK:=(FALSE);
            CRON[32].InitOK:=(FALSE);
            CRON[33].InitOK:=(FALSE);
            CRON[34].InitOK:=(FALSE);
            CRON[35].InitOK:=(FALSE);
            CRON[36].InitOK:=(FALSE);
            CRON[37].InitOK:=(FALSE);
            CRON[38].InitOK:=(FALSE);
        }
END_VISUALIZATION

